// Functions/Machine Learning/F_VN_CreateLbgModel

	{attribute 'TcIecLibraryType'}
	{attribute 'external_name' := 'F_VN_CreateLbgModel_GUID_C00C428F_55C9_4971_DE2F_CFD3295E8336'}
	(* Create a LBG model of the specified type. The initial reference count is set to one if a new model is created and kept, otherwise. Models of this type neither support on-line training (sample by sample) nor retraining. *)
	FUNCTION F_VN_CreateLbgModel : HRESULT
	VAR_INPUT
		ipMlModel	:	REFERENCE TO ITcVnMlModel;	(* Returns the created model (Non-zero interface pointers are reused.) *)
		eLbgType	:	ETcVnPrototypeClusterer;	(* LBG model type *)
		nMaxClusters	:	UDINT;	(* Maximum number of clusters *)
		fMaxClusterRadius	:	LREAL;	(* Maximum allowed radius (L2 norm) of a single cluster, i.e. clusters with a higher radius will be split into smaller ones, until a global number of nMaxClusters is reached. *)
		bSingleSplitSteps	:	BOOL;	(* If true, the global optimization is always run after a single cluster has been split. If false, several clusters are split within the same step before applying the global optimization. Applying the global optimization less often is faster, but can lead to less optimal results, especially having 2 nearby clusters that could be represented by 1. *)
		hrPrev	:	HRESULT;	(* HRESULT indicating the result of previous operations (If SUCCEEDED(hrPrev) equals false, no operation is executed.) *)
	END_VAR

END_FUNCTION

// Functions/Machine Learning/F_VN_CreateLbgModelExp

	{attribute 'TcIecLibraryType'}
	{attribute 'external_name' := 'F_VN_CreateLbgModelExp_GUID_151363FF_384A_48B1_E262_C0F66CE59E70'}
	(* Create a LBG model of the specified type. The initial reference count is set to one if a new model is created and kept, otherwise. Models of this type neither support on-line training (sample by sample) nor retraining. (expert function) *)
	FUNCTION F_VN_CreateLbgModelExp : HRESULT
	VAR_INPUT
		ipMlModel	:	REFERENCE TO ITcVnMlModel;	(* Returns the created model (Non-zero interface pointers are reused.) *)
		eLbgType	:	ETcVnPrototypeClusterer;	(* LBG model type *)
		nMaxClusters	:	UDINT;	(* Maximum number of clusters *)
		fMaxClusterRadius	:	LREAL;	(* Maximum allowed radius (L2 norm) of a single cluster, i.e. clusters with a higher radius will be split into smaller ones, until a global number of nMaxClusters is reached. *)
		bSingleSplitSteps	:	BOOL;	(* If true, the global optimization is always run after a single cluster has been split. If false, several clusters are split within the same step before applying the global optimization. Applying the global optimization less often is faster, but can lead to less optimal results, especially having 2 nearby clusters that could be represented by 1. *)
		bDoublePrecision	:	BOOL;	(* If true, the model is generated with double precision (LREAL) instead of single precision (REAL). (default: FALSE) *)
		nMaxIterations	:	UDINT;	(* Maximum number of iterations (triggers the usage of the default value of 10 if it equals 0) *)
		fEpsilon	:	LREAL;	(* Maximum allowed difference of the error between two successive iterations (triggers the usage of the default value of 0.001 if it equals 0) *)
		hrPrev	:	HRESULT;	(* HRESULT indicating the result of previous operations (If SUCCEEDED(hrPrev) equals false, no operation is executed.) *)
	END_VAR

END_FUNCTION

// Functions/Machine Learning/F_VN_CreateLdaTransform

	{attribute 'TcIecLibraryType'}
	{attribute 'external_name' := 'F_VN_CreateLdaTransform_GUID_D77D3FD7_41F4_408F_DD19_2A56BE0EA5DA'}
	(* Create an LDA-based feature transform from the provided data. The number of samples must be >= the number of features and the number of classes must be >= 2. The initial reference count is set to one if a new model is created and kept, otherwise. *)
	FUNCTION F_VN_CreateLdaTransform : HRESULT
	VAR_INPUT
		ipMlModel	:	REFERENCE TO ITcVnMlModel;	(* Returns the created feature transform (Non-zero interface pointers are reused.) *)
		ipSamples	:	ITcUnknown;	(* Container holding a batch of input samples (ContainerType_Vector_Vector_REAL or ContainerType_Vector_Vector_LREAL) *)
		ipClasses	:	ITcVnContainer;	(* Class labels corresponding to the input samples (ContainerType_Vector_DINT) *)
		hrPrev	:	HRESULT;	(* HRESULT indicating the result of previous operations (If SUCCEEDED(hrPrev) equals false, no operation is executed.) *)
	END_VAR

END_FUNCTION

// Functions/Machine Learning/F_VN_CreateLdaTransformViaComponentNum

	{attribute 'TcIecLibraryType'}
	{attribute 'external_name' := 'F_VN_CreateLdaTransformViaComponentNum_GUID_F3791234_4F92_4DC1_C9F2_B56383471767'}
	(* Create an LDA-based feature transform from the provided data where the number of components to be used is predefined. The number of samples must be >= the number of features and the number of classes must be >= 2. The initial reference count is set to one if a new model is created and kept, otherwise. (expert function) *)
	FUNCTION F_VN_CreateLdaTransformViaComponentNum : HRESULT
	VAR_INPUT
		ipMlModel	:	REFERENCE TO ITcVnMlModel;	(* Returns the created feature transform (Non-zero interface pointers are reused.) *)
		ipSamples	:	ITcUnknown;	(* Container holding a batch of input samples (ContainerType_Vector_Vector_REAL or ContainerType_Vector_Vector_LREAL) *)
		ipClasses	:	ITcVnContainer;	(* Class labels corresponding to the input samples (ContainerType_Vector_DINT) *)
		nComponentNum	:	UDINT;	(* Number of components (nComponentNum must be smaller than the number of classes. A value of 0 results in the automatic computation of the maximum number of components.) *)
		hrPrev	:	HRESULT;	(* HRESULT indicating the result of previous operations (If SUCCEEDED(hrPrev) equals false, no operation is executed.) *)
	END_VAR

END_FUNCTION

// Functions/Machine Learning/F_VN_CreateNbcModel

	{attribute 'TcIecLibraryType'}
	{attribute 'external_name' := 'F_VN_CreateNbcModel_GUID_B291926B_539A_480B_CC9D_93BEFD4CDD23'}
	(* Create a normal Bayes classifier of the specified type. The initial reference count is set to one if a new model is created and kept, otherwise. In order to train normal Bayes classifiers, a sufficiently high number of samples is required for each class. It depends on the number of features and the distribution of the data. Hence, it needs to be tested for each application. Models of this type do not support on-line training (sample by sample). For the retraining of such classifier models, the set of presented classes must be identical to the previous learning steps. Otherwise, an exception is raised. *)
	FUNCTION F_VN_CreateNbcModel : HRESULT
	VAR_INPUT
		ipMlModel	:	REFERENCE TO ITcVnMlModel;	(* Returns the created model (Non-zero interface pointers are reused.) *)
		eNbcType	:	ETcVnNbc;	(* Normal Bayes classifier type *)
		hrPrev	:	HRESULT;	(* HRESULT indicating the result of previous operations (If SUCCEEDED(hrPrev) equals false, no operation is executed.) *)
	END_VAR

END_FUNCTION

// Functions/Machine Learning/F_VN_CreatePcaTransform

	{attribute 'TcIecLibraryType'}
	{attribute 'external_name' := 'F_VN_CreatePcaTransform_GUID_B2B7912B_986F_4726_FAF9_1BE1D18B6FE5'}
	(* Create a PCA-based feature transform from the provided data. The maximum number of principal components that can be computed equals the minimum of the number of samples and the number of features. The initial reference count is set to one if a new model is created and kept, otherwise. *)
	FUNCTION F_VN_CreatePcaTransform : HRESULT
	VAR_INPUT
		ipMlModel	:	REFERENCE TO ITcVnMlModel;	(* Returns the created feature transform (Non-zero interface pointers are reused.) *)
		ipSamples	:	ITcUnknown;	(* Container holding a batch of input samples (ContainerType_Vector_Vector_REAL or ContainerType_Vector_Vector_LREAL) *)
		hrPrev	:	HRESULT;	(* HRESULT indicating the result of previous operations (If SUCCEEDED(hrPrev) equals false, no operation is executed.) *)
	END_VAR

END_FUNCTION

// Functions/Machine Learning/F_VN_CreatePcaTransformViaComponentNum

	{attribute 'TcIecLibraryType'}
	{attribute 'external_name' := 'F_VN_CreatePcaTransformViaComponentNum_GUID_40831A82_3642_480F_ED98_62DA272661FF'}
	(* Create a PCA-based feature transform from the provided data where the number of prinicpal components to be used is predefined. The maximum number of principal components that can be computed equals the minimum of the number of samples and the number of features. The initial reference count is set to one if a new model is created and kept, otherwise. (expert function) *)
	FUNCTION F_VN_CreatePcaTransformViaComponentNum : HRESULT
	VAR_INPUT
		ipMlModel	:	REFERENCE TO ITcVnMlModel;	(* Returns the created feature transform (Non-zero interface pointers are reused.) *)
		ipSamples	:	ITcUnknown;	(* Container holding a batch of input samples (ContainerType_Vector_Vector_REAL or ContainerType_Vector_Vector_LREAL) *)
		nComponentNum	:	UDINT;	(* Number of principal components (A value of 0 results in the automatic computation of the maximum number of components.) *)
		hrPrev	:	HRESULT;	(* HRESULT indicating the result of previous operations (If SUCCEEDED(hrPrev) equals false, no operation is executed.) *)
	END_VAR

END_FUNCTION

// Functions/Machine Learning/F_VN_CreatePcaTransformViaVariance

	{attribute 'TcIecLibraryType'}
	{attribute 'external_name' := 'F_VN_CreatePcaTransformViaVariance_GUID_7593ED13_6826_4CA8_C043_9ACE9956F61F'}
	(* Create a PCA-based feature transform from the provided data based on a given fraction of variance to be retained. The maximum number of principal components that can be computed equals the minimum of the number of samples and the number of features. The initial reference count is set to one if a new model is created and kept, otherwise. (expert function) *)
	FUNCTION F_VN_CreatePcaTransformViaVariance : HRESULT
	VAR_INPUT
		ipMlModel	:	REFERENCE TO ITcVnMlModel;	(* Returns the created feature transform (Non-zero interface pointers are reused.) *)
		ipSamples	:	ITcUnknown;	(* Container holding a batch of input samples (ContainerType_Vector_Vector_REAL or ContainerType_Vector_Vector_LREAL) *)
		fRetainedVariance	:	LREAL;	(* Fraction of variance that is to be retained by the PCA (A value of 1.0 signifies 100%.) *)
		hrPrev	:	HRESULT;	(* HRESULT indicating the result of previous operations (If SUCCEEDED(hrPrev) equals false, no operation is executed.) *)
	END_VAR

END_FUNCTION

// Functions/Machine Learning/F_VN_CreateRTreesModel

	{attribute 'TcIecLibraryType'}
	{attribute 'external_name' := 'F_VN_CreateRTreesModel_GUID_361E493C_0B92_4424_E04B_1ECB2685F6EE'}
	(* Create a random trees model of the specified type. The initial reference count is set to one if a new model is created and kept, otherwise. Models of this type neither support on-line training (sample by sample) nor retraining. Predictions can only be scalar. *)
	FUNCTION F_VN_CreateRTreesModel : HRESULT
	VAR_INPUT
		ipMlModel	:	REFERENCE TO ITcVnMlModel;	(* Returns the created model (Non-zero interface pointers are reused.) *)
		eRTreesType	:	ETcVnRTrees;	(* Random trees model type *)
		hrPrev	:	HRESULT;	(* HRESULT indicating the result of previous operations (If SUCCEEDED(hrPrev) equals false, no operation is executed.) *)
	END_VAR

END_FUNCTION

// Functions/Machine Learning/F_VN_CreateRTreesModelExp

	{attribute 'TcIecLibraryType'}
	{attribute 'external_name' := 'F_VN_CreateRTreesModelExp_GUID_DCAA6B97_3E63_4846_D44A_21B2790A7B88'}
	(* Create a random trees model of the specified type. The initial reference count is set to one if a new model is created and kept, otherwise. Models of this type neither support on-line training (sample by sample) nor retraining. Predictions can only be scalar. (expert function) *)
	FUNCTION F_VN_CreateRTreesModelExp : HRESULT
	VAR_INPUT
		ipMlModel	:	REFERENCE TO ITcVnMlModel;	(* Returns the created model (Non-zero interface pointers are reused.) *)
		eRTreesType	:	ETcVnRTrees;	(* Random trees model type *)
		nMaxDepth	:	UDINT;	(* Maximum tree depth (default: 5) *)
		nMinSamples	:	UDINT;	(* Minimum number of samples within a node required for splitting (default: 10) *)
		nActiveVariables	:	UDINT;	(* Number of variables considered for splitting (0 means sqrt(total number of variables); default: 0) *)
		nMaxIterations	:	UDINT;	(* Maximum number of iterations (disabled if it equals 0 and fEpsilon is different from 0.0; triggers the usage of the default value of 50 if nMaxIterations and fEpsilon equal 0) *)
		fEpsilon	:	LREAL;	(* Maximum allowed difference of the error between two successive iterations (disabled if it equals 0.0 and nMaxIterations is different from 0; triggers the usage of the default value of 0.1 if nMaxIterations and fEpsilon equal 0) *)
		hrPrev	:	HRESULT;	(* HRESULT indicating the result of previous operations (If SUCCEEDED(hrPrev) equals false, no operation is executed.) *)
	END_VAR

END_FUNCTION

// Functions/Machine Learning/F_VN_CreateRTreesModelExp2

	{attribute 'TcIecLibraryType'}
	{attribute 'external_name' := 'F_VN_CreateRTreesModelExp2_GUID_A3B951DB_7DFC_4984_C9A1_23F5FD764134'}
	(* Create a random trees model of the specified type. The initial reference count is set to one if a new model is created and kept, otherwise. Models of this type neither support on-line training (sample by sample) nor retraining. Predictions can only be scalar. (expert function) *)
	FUNCTION F_VN_CreateRTreesModelExp2 : HRESULT
	VAR_INPUT
		ipMlModel	:	REFERENCE TO ITcVnMlModel;	(* Returns the created model (Non-zero interface pointers are reused.) *)
		eRTreesType	:	ETcVnRTrees;	(* Random trees model type *)
		nMaxDepth	:	UDINT;	(* Maximum tree depth (default: 5) *)
		nMinSamples	:	UDINT;	(* Minimum number of samples within a node required for splitting (default: 10) *)
		nActiveVariables	:	UDINT;	(* Number of variables considered for splitting (0 means sqrt(total number of variables); default: 0) *)
		nMaxIterations	:	UDINT;	(* Maximum number of iterations (disabled if it equals 0 and fEpsilon is different from 0.0; triggers the usage of the default value of 50 if nMaxIterations and fEpsilon equal 0) *)
		fEpsilon	:	LREAL;	(* Maximum allowed difference of the error between two successive iterations (disabled if it equals 0.0 and nMaxIterations is different from 0; triggers the usage of the default value of 0.1 if nMaxIterations and fEpsilon equal 0) *)
		fRegressionAccuracy	:	REAL;	(* Termination criterion for regressors (only for regressors; set to default if not allowed; default: 0.0) *)
		ipClassPriors	:	ITcVnContainer;	(* Class priors (ContainerType_Vector_REAL or ContainerType_Vector_LREAL; only for classifiers; optional, set to 0 if not required or not allowed; default: 0) *)
		hrPrev	:	HRESULT;	(* HRESULT indicating the result of previous operations (If SUCCEEDED(hrPrev) equals false, no operation is executed.) *)
	END_VAR

END_FUNCTION

// Functions/Machine Learning/F_VN_CreateStaModel

	{attribute 'TcIecLibraryType'}
	{attribute 'external_name' := 'F_VN_CreateStaModel_GUID_0E65F544_36C9_4DC3_E430_89B77157AED0'}
	(* Create a Simplified TopoART neural network of the specified type. The initial reference count is set to one if a new model is created and kept, otherwise. Models of this type support on-line training (sample by sample), retraining, as well as scalar and vectorial predictions. It requires all input except class labels (i.e., samples and training outputs/predictions) to lie in the interval [0.0, 1.0]. The predictions of regressors need to be rescaled from the interval [0.0, 1.0] to their respective value range before usage. Depending on the parameter settings and the number of available training samples, repeated training with the same data may improve the results. Like other neural networks based on the Adaptive Resonance Theory (ART), Simplified TopoART neural networks are not prone to catastrophic inference and patricularly well-suited to incremental learning tasks. *)
	FUNCTION F_VN_CreateStaModel : HRESULT
	VAR_INPUT
		ipMlModel	:	REFERENCE TO ITcVnMlModel;	(* Returns the created model (Non-zero interface pointers are reused.) *)
		eStaType	:	ETcVnSta;	(* Simpified TopoART model type *)
		fRho	:	LREAL;	(* Vigilance parameter (controls the number of neurons that are inserted and the maximum size of the formed categories; valid range: [0.0, 1.0]; suggested range: [0.8, 1.0)) *)
		hrPrev	:	HRESULT;	(* HRESULT indicating the result of previous operations (If SUCCEEDED(hrPrev) equals false, no operation is executed.) *)
	END_VAR

END_FUNCTION

// Functions/Machine Learning/F_VN_CreateStaModelExp

	{attribute 'TcIecLibraryType'}
	{attribute 'external_name' := 'F_VN_CreateStaModelExp_GUID_60C95C96_C531_4303_F18A_D4FE39CB265F'}
	(* Create a Simplified TopoART neural network of the specified type. The initial reference count is set to one if a new model is created and kept, otherwise. Models of this type support on-line training (sample by sample), retraining, as well as scalar and vectorial predictions. It requires all input except class labels (i.e., samples and training outputs/predictions) to lie in the interval [0.0, 1.0]. The predictions of regressors need to be rescaled from the interval [0.0, 1.0] to their respective value range before usage. Depending on the parameter settings and the number of available training samples, repeated training with the same data may improve the results. Like other neural networks based on the Adaptive Resonance Theory (ART), Simplified TopoART neural networks are not prone to catastrophic inference and patricularly well-suited to incremental learning tasks. (expert function) *)
	FUNCTION F_VN_CreateStaModelExp : HRESULT
	VAR_INPUT
		ipMlModel	:	REFERENCE TO ITcVnMlModel;	(* Returns the created model (Non-zero interface pointers are reused.) *)
		eStaType	:	ETcVnSta;	(* Simpified TopoART model type *)
		fRho	:	LREAL;	(* Vigilance parameter (controls the number of neurons that are inserted and the maximum size of the formed categories; valid range: [0.0, 1.0]; suggested range: [0.8, 1.0)) *)
		nNu	:	UDINT;	(* Number of neurons used for classification and prediction (must be larger than or equal to 1; suggested range: [1, 10); default: 3) *)
		bDoublePrecision	:	BOOL;	(* If true, the model is generated with double precision (LREAL) instead of single precision (REAL). (default: FALSE) *)
		hrPrev	:	HRESULT;	(* HRESULT indicating the result of previous operations (If SUCCEEDED(hrPrev) equals false, no operation is executed.) *)
	END_VAR

END_FUNCTION

// Functions/Machine Learning/F_VN_CreateStaModelExp2

	{attribute 'TcIecLibraryType'}
	{attribute 'external_name' := 'F_VN_CreateStaModelExp2_GUID_DC5ABDD2_E185_452E_E9B5_8EF979CD80B8'}
	(* Create a Simplified TopoART neural network of the specified type. The initial reference count is set to one if a new model is created and kept, otherwise. Models of this type support on-line training (sample by sample), retraining, as well as scalar and vectorial predictions. It requires all input except class labels (i.e., samples and training outputs/predictions) to lie in the interval [0.0, 1.0]. The predictions of regressors need to be rescaled from the interval [0.0, 1.0] to their respective value range before usage. Depending on the parameter settings and the number of available training samples, repeated training with the same data may improve the results. Like other neural networks based on the Adaptive Resonance Theory (ART), Simplified TopoART neural networks are not prone to catastrophic inference and patricularly well-suited to incremental learning tasks. (additional expert function providing parameters for fine-tuning and noise reduction) *)
	FUNCTION F_VN_CreateStaModelExp2 : HRESULT
	VAR_INPUT
		ipMlModel	:	REFERENCE TO ITcVnMlModel;	(* Returns the created model (Non-zero interface pointers are reused.) *)
		eStaType	:	ETcVnSta;	(* Simpified TopoART model type *)
		fRho	:	LREAL;	(* Vigilance parameter (controls the number of neurons that are inserted and the maximum size of the formed categories; valid range: [0.0, 1.0]; suggested range: [0.8, 1.0)) *)
		nNu	:	UDINT;	(* Number of neurons used for classification and prediction (must be larger than or equal to 1; suggested range: [1, 10); default: 3) *)
		bDoublePrecision	:	BOOL;	(* If true, the model is generated with double precision (LREAL) instead of single precision (REAL). (default: FALSE) *)
		fBetaSbm	:	LREAL;	(* Learning rate of the second best-matching neuron (learning the second best-matching neuron keeps related categories closer together and might improve the results but may require a higher number of neurons and training runs; a value of 0.0 disables learning of the second best-matching neuron; valid range: [0.0, 1.0]; suggested range: [0.0, 0.5]); default: 0.0 *)
		nPhi	:	UDINT;	(* Number of samples a neuron must have learnt to become permanent (required for noise reduction; works in conjunction with nTau; must be larger than or equal to 1; higher values intensify noise reduction; a value of 1 disables removal of neuron candidates; default: 1) *)
		nTau	:	UDINT;	(* Number of learning steps after which node removal is performed (required for noise reduction; works in conjunction with nPhi; must be large enough to allow neuron candidates representing non-noise samples to become the best-matching neuron at least nPhi times before node removal; default: 100) *)
		hrPrev	:	HRESULT;	(* HRESULT indicating the result of previous operations (If SUCCEEDED(hrPrev) equals false, no operation is executed.) *)
	END_VAR

END_FUNCTION

// Functions/Machine Learning/F_VN_CreateSvmModel

	{attribute 'TcIecLibraryType'}
	{attribute 'external_name' := 'F_VN_CreateSvmModel_GUID_6608170F_8E55_4CB7_CA5D_A5F69CCA9D00'}
	(* Create an SVM model of the specified type. The initial reference count is set to one if a new model is created and kept, otherwise. Models of this type neither support on-line training (sample by sample) nor retraining. Predictions can only be scalar. *)
	FUNCTION F_VN_CreateSvmModel : HRESULT
	VAR_INPUT
		ipMlModel	:	REFERENCE TO ITcVnMlModel;	(* Returns the created model (Non-zero interface pointers are reused.) *)
		eSvmType	:	ETcVnSvm;	(* SVM model type *)
		fC	:	LREAL;	(* Parameter C (required for TCVN_SVM_C_CLASSIFIER, TCVN_SVM_EPS_REGRESSOR, and TCVN_SVM_NU_REGRESSOR; ignored otherwise) *)
		fNu	:	LREAL;	(* Parameter nu (required for TCVN_SVM_NU_CLASSIFIER, TCVN_SVM_NOVELTY_DETECTOR, and TCVN_SVM_NU_REGRESSOR; ignored otherwise) *)
		fP	:	LREAL;	(* Parameter p (required for TCVN_SVM_EPS_REGRESSOR; ignored otherwise) *)
		eKernelType	:	ETcVnSvmKernelType;	(* Kernel type *)
		fGamma	:	LREAL;	(* Parameter gamma (used by polynomial, RBF, sigmoid, and chi-squared kernels; ignored otherwise) *)
		fCoef0	:	LREAL;	(* parameter coef0 (used by polynomial and sigmoid kernels; ignored otherwise) *)
		fDegree	:	LREAL;	(* Degree (used by polynomial kernels; ignored otherwise) *)
		hrPrev	:	HRESULT;	(* HRESULT indicating the result of previous operations (If SUCCEEDED(hrPrev) equals false, no operation is executed.) *)
	END_VAR

END_FUNCTION

// Functions/Machine Learning/F_VN_CreateSvmModelExp

	{attribute 'TcIecLibraryType'}
	{attribute 'external_name' := 'F_VN_CreateSvmModelExp_GUID_6B1D8D00_DDAB_4438_FB92_B0FDD976C945'}
	(* Create an SVM model of the specified type. The initial reference count is set to one if a new model is created and kept, otherwise. Models of this type neither support on-line training (sample by sample) nor retraining. Predictions can only be scalar. (expert function) *)
	FUNCTION F_VN_CreateSvmModelExp : HRESULT
	VAR_INPUT
		ipMlModel	:	REFERENCE TO ITcVnMlModel;	(* Returns the created model (Non-zero interface pointers are reused.) *)
		eSvmType	:	ETcVnSvm;	(* SVM model type *)
		fC	:	LREAL;	(* Parameter C (required for TCVN_SVM_C_CLASSIFIER, TCVN_SVM_EPS_REGRESSOR, and TCVN_SVM_NU_REGRESSOR; ignored otherwise) *)
		fNu	:	LREAL;	(* Parameter nu (required for TCVN_SVM_NU_CLASSIFIER, TCVN_SVM_NOVELTY_DETECTOR, and TCVN_SVM_NU_REGRESSOR; ignored otherwise) *)
		fP	:	LREAL;	(* Parameter p (required for TCVN_SVM_EPS_REGRESSOR; ignored otherwise) *)
		eKernelType	:	ETcVnSvmKernelType;	(* Kernel type *)
		fGamma	:	LREAL;	(* Parameter gamma (used by polynomial, RBF, sigmoid, and chi-squared kernels; ignored otherwise) *)
		fCoef0	:	LREAL;	(* Parameter coef0 (used by polynomial and sigmoid kernels; ignored otherwise) *)
		fDegree	:	LREAL;	(* Degree (used by polynomial kernels; ignored otherwise) *)
		nMaxIterations	:	UDINT;	(* Maximum number of iterations (disabled if it equals 0 and fEpsilon is different from 0.0; triggers the usage of the default value of 100000 if nMaxIterations and fEpsilon equal 0) *)
		fEpsilon	:	LREAL;	(* Maximum allowed difference of the error between two successive iterations (disabled if it equals 0.0 and nMaxIterations is different from 0; triggers the usage of the default value of 0.00001 if nMaxIterations and fEpsilon equal 0) *)
		hrPrev	:	HRESULT;	(* HRESULT indicating the result of previous operations (If SUCCEEDED(hrPrev) equals false, no operation is executed.) *)
	END_VAR

END_FUNCTION

// Functions/Machine Learning/F_VN_CreateSvmModelExp2

	{attribute 'TcIecLibraryType'}
	{attribute 'external_name' := 'F_VN_CreateSvmModelExp2_GUID_6FD5F0B0_2D5E_4EC3_E8E4_B31A19CD0010'}
	(* Create an SVM model of the specified type. The initial reference count is set to one if a new model is created and kept, otherwise. Models of this type neither support on-line training (sample by sample) nor retraining. Predictions can only be scalar. (additional expert function for C support vector classifiers) *)
	FUNCTION F_VN_CreateSvmModelExp2 : HRESULT
	VAR_INPUT
		ipMlModel	:	REFERENCE TO ITcVnMlModel;	(* Returns the created model (Non-zero interface pointers are reused.) *)
		eSvmType	:	ETcVnSvm;	(* SVM model type *)
		fC	:	LREAL;	(* Parameter C (required for TCVN_SVM_C_CLASSIFIER, TCVN_SVM_EPS_REGRESSOR, and TCVN_SVM_NU_REGRESSOR; ignored otherwise) *)
		fNu	:	LREAL;	(* Parameter nu (required for TCVN_SVM_NU_CLASSIFIER, TCVN_SVM_NOVELTY_DETECTOR, and TCVN_SVM_NU_REGRESSOR; ignored otherwise) *)
		fP	:	LREAL;	(* Parameter p (required for TCVN_SVM_EPS_REGRESSOR; ignored otherwise) *)
		eKernelType	:	ETcVnSvmKernelType;	(* Kernel type *)
		fGamma	:	LREAL;	(* Parameter gamma (used by polynomial, RBF, sigmoid, and chi-squared kernels; ignored otherwise) *)
		fCoef0	:	LREAL;	(* Parameter coef0 (used by polynomial and sigmoid kernels; ignored otherwise) *)
		fDegree	:	LREAL;	(* Degree (used by polynomial kernels; ignored otherwise) *)
		nMaxIterations	:	UDINT;	(* Maximum number of iterations (disabled if it equals 0 and fEpsilon is different from 0.0; triggers the usage of the default value of 100000 if nMaxIterations and fEpsilon equal 0) *)
		fEpsilon	:	LREAL;	(* Maximum allowed difference of the error between two successive iterations (disabled if it equals 0.0 and nMaxIterations is different from 0; triggers the usage of the default value of 0.00001 if nMaxIterations and fEpsilon equal 0) *)
		ipClassWeights	:	ITcVnContainer;	(* Class weights (ContainerType_Vector_REAL or ContainerType_Vector_LREAL; only valid if eSvmType equals TCVN_SVM_C_CLASSIFIER; optional, set to 0 if not required or not allowed; default: 0) *)
		hrPrev	:	HRESULT;	(* HRESULT indicating the result of previous operations (If SUCCEEDED(hrPrev) equals false, no operation is executed.) *)
	END_VAR

END_FUNCTION

// Functions/Machine Learning/F_VN_CreateSvmSgdClassifier

	{attribute 'TcIecLibraryType'}
	{attribute 'external_name' := 'F_VN_CreateSvmSgdClassifier_GUID_C9EE268D_C05A_48F3_D32E_D9B3E0FBCDCB'}
	(* Create a linear SVM classifier using stochastic gradient descent for training. The initial reference count is set to one if a new model is created and kept, otherwise. This SVM classifier is only applicable to binary classification problems. It learns a separating hyperplane between a class with label -1 and a class with label 1. These class labels are predefined. For training, any positive class labels are mapped to 1 and any negative class labels are mapped to -1. Models of this type neither support on-line training (sample by sample) nor retraining. *)
	FUNCTION F_VN_CreateSvmSgdClassifier : HRESULT
	VAR_INPUT
		ipMlModel	:	REFERENCE TO ITcVnMlModel;	(* Returns the created model (Non-zero interface pointers are reused.) *)
		hrPrev	:	HRESULT;	(* HRESULT indicating the result of previous operations (If SUCCEEDED(hrPrev) equals false, no operation is executed.) *)
	END_VAR

END_FUNCTION

// Functions/Machine Learning/F_VN_CreateSvmSgdClassifierExp

	{attribute 'TcIecLibraryType'}
	{attribute 'external_name' := 'F_VN_CreateSvmSgdClassifierExp_GUID_35712FDB_BBEA_4B29_FC4D_61FC511DA0EB'}
	(* Create a linear SVM classifier using stochastic gradient descent for training. The initial reference count is set to one if a new model is created and kept, otherwise. This SVM classifier is only applicable to binary classification problems. It learns a separating hyperplane between a class with label -1 and a class with label 1. These class labels are predefined. For training, any positive class labels are mapped to 1 and any negative class labels are mapped to -1. Models of this type neither support on-line training (sample by sample) nor retraining. (expert function) *)
	FUNCTION F_VN_CreateSvmSgdClassifierExp : HRESULT
	VAR_INPUT
		ipMlModel	:	REFERENCE TO ITcVnMlModel;	(* Returns the created model (Non-zero interface pointers are reused.) *)
		eType	:	ETcVnSvmSgdClassifierType;	(* Learning algorithm type (default: TCVN_SSCT_ASGD) *)
		eMarginType	:	ETcVnSvmSgdClassifierMarginType;	(* Margin type (default: TCVN_SSCMT_SOFT_MARGIN) *)
		fMarginRegularization	:	REAL;	(* Margin regularization parameter (default: 0.00001) *)
		fInitialStepSize	:	REAL;	(* Initial step size (default: 0.05) *)
		fStepDecreasingPower	:	REAL;	(* Power parameter (default: 0.75) *)
		nMaxIterations	:	UDINT;	(* Maximum number of iterations (disabled if it equals 0 and fEpsilon is different from 0.0; triggers the usage of the default value of 100000 if nMaxIterations and fEpsilon equal 0) *)
		fEpsilon	:	LREAL;	(* Maximum allowed difference of the error between two successive iterations (disabled if it equals 0.0 and nMaxIterations is different from 0; triggers the usage of the default value of 0.00001 if nMaxIterations and fEpsilon equal 0) *)
		hrPrev	:	HRESULT;	(* HRESULT indicating the result of previous operations (If SUCCEEDED(hrPrev) equals false, no operation is executed.) *)
	END_VAR

END_FUNCTION

// Functions/Machine Learning/F_VN_FeatureTransform

	{attribute 'TcIecLibraryType'}
	{attribute 'external_name' := 'F_VN_FeatureTransform_GUID_C607A85C_BB4D_46AF_DE31_007EC6E109EA'}
	(* Apply a feature transform to one or more sample(s). *)
	FUNCTION F_VN_FeatureTransform : HRESULT
	VAR_INPUT
		ipFeatureTransform	:	ITcVnMlModel;	(* Feature transform instance to be used *)
		ipSamples	:	ITcUnknown;	(* Container holding one or more of input sample(s) (ContainerType_Vector_REAL, ContainerType_Vector_LREAL, ContainerType_Vector_Vector_REAL, or ContainerType_Vector_Vector_LREAL) *)
		pipTransformed	:	POINTER TO ITcUnknown;	(* Returns the transformed sample(s) using the same type like ipSamples *)
		hrPrev	:	HRESULT;	(* HRESULT indicating the result of previous operations (If SUCCEEDED(hrPrev) equals false, no operation is executed.) *)
	END_VAR

END_FUNCTION

// Functions/Machine Learning/F_VN_GetBatchClusters

	{attribute 'TcIecLibraryType'}
	{attribute 'external_name' := 'F_VN_GetBatchClusters_GUID_528E2B3F_88E6_4E83_EA33_7AE81270B54C'}
	(* Get the IDs of the best-matching clusters of a batch of samples. *)
	FUNCTION F_VN_GetBatchClusters : HRESULT
	VAR_INPUT
		ipClusterer	:	ITcVnMlModel;	(* Clusterer to be used *)
		ipSamples	:	ITcUnknown;	(* Container holding a batch of input samples (ContainerType_Vector_Vector_REAL or ContainerType_Vector_Vector_LREAL) *)
		ipClusters	:	REFERENCE TO ITcVnContainer;	(* Returns the cluster IDs (ContainerType_Vector_DINT) *)
		hrPrev	:	HRESULT;	(* HRESULT indicating the result of previous operations (If SUCCEEDED(hrPrev) equals false, no operation is executed.) *)
	END_VAR

END_FUNCTION

// Functions/Machine Learning/F_VN_GetBatchClustersExp

	{attribute 'TcIecLibraryType'}
	{attribute 'external_name' := 'F_VN_GetBatchClustersExp_GUID_EA27BC56_5775_49D6_D10F_C11E25D16558'}
	(* Get the IDs of the best-matching clusters of a batch of samples. *)
	FUNCTION F_VN_GetBatchClustersExp : HRESULT
	VAR_INPUT
		ipClusterer	:	ITcVnMlModel;	(* Clusterer to be used *)
		ipSamples	:	ITcUnknown;	(* Container holding a batch of input samples (ContainerType_Vector_Vector_REAL or ContainerType_Vector_Vector_LREAL) *)
		ipClusters	:	REFERENCE TO ITcVnContainer;	(* Returns the cluster IDs (ContainerType_Vector_DINT) *)
		ipNovelties	:	REFERENCE TO ITcVnContainer;	(* Returns the degree of novelty (0.0 if a sample is completely known; > 0.0 otherwise) of each sample (ContainerType_Vector_REAL; optional, set to 0 if not required) *)
		hrPrev	:	HRESULT;	(* HRESULT indicating the result of previous operations (If SUCCEEDED(hrPrev) equals false, no operation is executed.) *)
	END_VAR

END_FUNCTION

// Functions/Machine Learning/F_VN_GetBatchNovelties

	{attribute 'TcIecLibraryType'}
	{attribute 'external_name' := 'F_VN_GetBatchNovelties_GUID_7C3BAC31_B33D_4380_E65E_AEEC8DBAEDE0'}
	(* Get the degree of novelty of multiple samples. *)
	FUNCTION F_VN_GetBatchNovelties : HRESULT
	VAR_INPUT
		ipNoveltyDetector	:	ITcVnMlModel;	(* Novelty detector to be used *)
		ipSamples	:	ITcUnknown;	(* Container holding a batch of input samples (ContainerType_Vector_Vector_REAL or ContainerType_Vector_Vector_LREAL) *)
		ipNovelties	:	REFERENCE TO ITcVnContainer;	(* Returns the degree of novelty (0.0 if a sample is completely known; > 0.0 otherwise) of each sample (ContainerType_Vector_REAL) *)
		hrPrev	:	HRESULT;	(* HRESULT indicating the result of previous operations (If SUCCEEDED(hrPrev) equals false, no operation is executed.) *)
	END_VAR

END_FUNCTION

// Functions/Machine Learning/F_VN_GetClusterCenter

	{attribute 'TcIecLibraryType'}
	{attribute 'external_name' := 'F_VN_GetClusterCenter_GUID_0F8CBC11_259F_42B1_EE6F_9AD92F7A06AE'}
	(* Get the center of a cluster. *)
	FUNCTION F_VN_GetClusterCenter : HRESULT
	VAR_INPUT
		ipClusterer	:	ITcVnMlModel;	(* Clusterer to be used *)
		nCluster	:	DINT;	(* Cluster ID of the cluster the center of which is requested *)
		ipCenter	:	REFERENCE TO ITcVnContainer;	(* Returns the cluster center (ContainerType_Vector_REAL or ContainerType_Vector_LREAL depending on the floating point type internally used by the clusterer) *)
		hrPrev	:	HRESULT;	(* HRESULT indicating the result of previous operations (If SUCCEEDED(hrPrev) equals false, no operation is executed.) *)
	END_VAR

END_FUNCTION

// Functions/Machine Learning/F_VN_GetClusterNum

	{attribute 'TcIecLibraryType'}
	{attribute 'external_name' := 'F_VN_GetClusterNum_GUID_548F7E1B_5B12_494E_CC7F_3482B1B8572D'}
	(* Get the number of clusters used by this clusterer. *)
	FUNCTION F_VN_GetClusterNum : HRESULT
	VAR_INPUT
		ipClusterer	:	ITcVnMlModel;	(* Clusterer to be used *)
	END_VAR
	VAR_IN_OUT
		nClusterNum	:	ULINT;	(* Returns the number of clusters *)
	END_VAR
	VAR_INPUT
		hrPrev	:	HRESULT;	(* HRESULT indicating the result of previous operations (If SUCCEEDED(hrPrev) equals false, no operation is executed.) *)
	END_VAR

END_FUNCTION

// Functions/Machine Learning/F_VN_GetFeatureScales

	{attribute 'TcIecLibraryType'}
	{attribute 'external_name' := 'F_VN_GetFeatureScales_GUID_FE369AE1_304E_4286_ECEF_EB86184B6B22'}
	(* Calculate the scaling parameters for each feature in the input samples based on the scaling type. *)
	FUNCTION F_VN_GetFeatureScales : HRESULT
	VAR_INPUT
		ipSamples	:	ITcVnContainer;	(* Container holding input sample(s) (ContainerType_Vector_REAL, ContainerType_Vector_LREAL, ContainerType_Vector_Vector_REAL or ContainerType_Vector_Vector_LREAL) *)
		ipScales	:	REFERENCE TO ITcVnContainer;	(* Returns a container with the scaling parameters for each feature (Vector_REAL or Vector_LREAL depending on the type of ipSamples). *)
		eFeatureScalingType	:	ETcVnFeatureScalingType;	(* Feature scaling type *)
		hrPrev	:	HRESULT;	(* HRESULT indicating the result of previous operations (If SUCCEEDED(hrPrev) equals false, no operation is executed.) *)
	END_VAR

END_FUNCTION

// Functions/Machine Learning/F_VN_GetSampleCluster

	{attribute 'TcIecLibraryType'}
	{attribute 'external_name' := 'F_VN_GetSampleCluster_GUID_32F204F3_A186_4B1B_F32F_2AD94C5430BB'}
	(* Get the ID of the best-matching cluster of a single sample. *)
	FUNCTION F_VN_GetSampleCluster : HRESULT
	VAR_INPUT
		ipClusterer	:	ITcVnMlModel;	(* Clusterer to be used *)
		ipSample	:	ITcUnknown;	(* Container holding a single input sample (ContainerType_Vector_REAL or ContainerType_Vector_LREAL) *)
	END_VAR
	VAR_IN_OUT
		nCluster	:	DINT;	(* Returns the ID of the cluster the sample has been assigned to *)
	END_VAR
	VAR_INPUT
		hrPrev	:	HRESULT;	(* HRESULT indicating the result of previous operations (If SUCCEEDED(hrPrev) equals false, no operation is executed.) *)
	END_VAR

END_FUNCTION

// Functions/Machine Learning/F_VN_GetSampleClusterExp

	{attribute 'TcIecLibraryType'}
	{attribute 'external_name' := 'F_VN_GetSampleClusterExp_GUID_3477724D_EC43_4000_ECAE_3FA8E7C5B7E6'}
	(* Get the ID of the best-matching cluster of a single sample. (expert function) *)
	FUNCTION F_VN_GetSampleClusterExp : HRESULT
	VAR_INPUT
		ipClusterer	:	ITcVnMlModel;	(* Clusterer to be used *)
		ipSample	:	ITcUnknown;	(* Container holding a single input sample (ContainerType_Vector_REAL or ContainerType_Vector_LREAL) *)
	END_VAR
	VAR_IN_OUT
		nCluster	:	DINT;	(* Returns the ID of the cluster the sample has been assigned to *)
	END_VAR
	VAR_INPUT
		fNovelty	:	REFERENCE TO REAL;	(* Returns the degree of novelty (0.0 if a sample is completely known; > 0.0 otherwise) of the presented sample (optional, set to 0 if not required) *)
		hrPrev	:	HRESULT;	(* HRESULT indicating the result of previous operations (If SUCCEEDED(hrPrev) equals false, no operation is executed.) *)
	END_VAR

END_FUNCTION

// Functions/Machine Learning/F_VN_GetSampleNovelty

	{attribute 'TcIecLibraryType'}
	{attribute 'external_name' := 'F_VN_GetSampleNovelty_GUID_D2B7DAC3_715A_4874_EE3F_A314571BD5C4'}
	(* Get the degree of novelty of a single sample. *)
	FUNCTION F_VN_GetSampleNovelty : HRESULT
	VAR_INPUT
		ipNoveltyDetector	:	ITcVnMlModel;	(* Novelty detector to be used *)
		ipSample	:	ITcUnknown;	(* Container holding a single input sample (ContainerType_Vector_REAL or ContainerType_Vector_LREAL) *)
	END_VAR
	VAR_IN_OUT
		fNovelty	:	REAL;	(* Returns the degree of novelty (0.0 if a sample is completely known; > 0.0 otherwise) of the presented sample *)
	END_VAR
	VAR_INPUT
		hrPrev	:	HRESULT;	(* HRESULT indicating the result of previous operations (If SUCCEEDED(hrPrev) equals false, no operation is executed.) *)
	END_VAR

END_FUNCTION

// Functions/Machine Learning/F_VN_InverseFeatureScaling

	{attribute 'TcIecLibraryType'}
	{attribute 'external_name' := 'F_VN_InverseFeatureScaling_GUID_15907737_CCFF_4C4C_EA62_BDD72702354F'}
	(* Apply the inverse of feature scaling to one or more sample(s). *)
	FUNCTION F_VN_InverseFeatureScaling : HRESULT
	VAR_INPUT
		ipSamples	:	ITcVnContainer;	(* Container holding one or more input sample(s) (ContainerType_Vector_REAL, ContainerType_Vector_LREAL, ContainerType_Vector_Vector_REAL, or ContainerType_Vector_Vector_LREAL) *)
		ipScales	:	ITcVnContainer;	(* Container with the scaling parameters of each feature (type ContainerType_Vector_REAL or ContainerType_Vector_LREAL). *)
		ipInverseSamples	:	REFERENCE TO ITcVnContainer;	(* Returns the inversed sample(s) using the scaling type and parameters of ipScales. It has the same type of ipSamples. If the same container ipSamples is used, the source data will be replaced. *)
		hrPrev	:	HRESULT;	(* HRESULT indicating the result of previous operations (If SUCCEEDED(hrPrev) equals false, no operation is executed.) *)
	END_VAR

END_FUNCTION

// Functions/Machine Learning/F_VN_InverseFeatureScaling_REAL

	{attribute 'TcIecLibraryType'}
	{attribute 'external_name' := 'F_VN_InverseFeatureScaling_REAL_GUID_F91E68ED_D57C_4247_F2CE_BAB31E6A8058'}
	(* Apply the inverse of feature scaling to a single value. *)
	FUNCTION F_VN_InverseFeatureScaling_REAL : HRESULT
	VAR_INPUT
		fSample	:	REAL;	(* Sample value *)
		ipScales	:	ITcVnContainer;	(* Container with the scaling parameters of each feature (type ContainerType_Vector_REAL or ContainerType_Vector_LREAL). *)
	END_VAR
	VAR_IN_OUT
		fInverseSample	:	REAL;	(* Returns the inversed sample. *)
	END_VAR
	VAR_INPUT
		hrPrev	:	HRESULT;	(* HRESULT indicating the result of previous operations (If SUCCEEDED(hrPrev) equals false, no operation is executed.) *)
	END_VAR

END_FUNCTION

// Functions/Machine Learning/F_VN_InverseFeatureScalingExp

	{attribute 'TcIecLibraryType'}
	{attribute 'external_name' := 'F_VN_InverseFeatureScalingExp_GUID_8B0E0F8E_1465_40CF_D892_BBD7360C8D03'}
	(* Apply the inverse of feature scaling to one or more sample(s). [fA, fB] should be used if the scaling has been performed using TCVN_FST1_MINMAX with a predetermined output range.. (expert function) *)
	FUNCTION F_VN_InverseFeatureScalingExp : HRESULT
	VAR_INPUT
		ipSamples	:	ITcVnContainer;	(* Container holding one or more input sample(s) (ContainerType_Vector_REAL, ContainerType_Vector_LREAL, ContainerType_Vector_Vector_REAL, or ContainerType_Vector_Vector_LREAL) *)
		ipScales	:	ITcVnContainer;	(* Container with the scaling parameters of each feature (type ContainerType_Vector_REAL or ContainerType_Vector_LREAL). *)
		ipInverseSamples	:	REFERENCE TO ITcVnContainer;	(* Returns the inversed sample(s) using the scaling type and parameters of ipScales. It has the same type of ipSamples. If the same container ipSamples is used, the source data will be replaced. *)
		fA	:	LREAL;	(* represents the lower bound of the range for TCVN_FST1_MINMAX *)
		fB	:	LREAL;	(* represents the upper bound of the range for TCVN_FST1_MINMAX *)
		hrPrev	:	HRESULT;	(* HRESULT indicating the result of previous operations (If SUCCEEDED(hrPrev) equals false, no operation is executed.) *)
	END_VAR

END_FUNCTION

// Functions/Machine Learning/F_VN_InverseFeatureScalingExp_REAL

	{attribute 'TcIecLibraryType'}
	{attribute 'external_name' := 'F_VN_InverseFeatureScalingExp_REAL_GUID_22A89423_ED3D_4292_D684_932CEE57D3B8'}
	(* Apply the inverse of feature scaling to a single value. [fA, fB] should be used if the scaling has been performed using TCVN_FST1_MINMAX with a predetermined output range. *)
	FUNCTION F_VN_InverseFeatureScalingExp_REAL : HRESULT
	VAR_INPUT
		fSample	:	REAL;	(* Sample value *)
		ipScales	:	ITcVnContainer;	(* Container with the scaling parameters of each feature (type ContainerType_Vector_REAL or ContainerType_Vector_LREAL). *)
	END_VAR
	VAR_IN_OUT
		fInverseSample	:	REAL;	(* Returns the inversed sample. *)
	END_VAR
	VAR_INPUT
		fA	:	LREAL;	(* represents the lower bound of the range for TCVN_FST1_MINMAX *)
		fB	:	LREAL;	(* represents the upper bound of the range for TCVN_FST1_MINMAX *)
		hrPrev	:	HRESULT;	(* HRESULT indicating the result of previous operations (If SUCCEEDED(hrPrev) equals false, no operation is executed.) *)
	END_VAR

END_FUNCTION

// Functions/Machine Learning/F_VN_InverseFeatureTransform

	{attribute 'TcIecLibraryType'}
	{attribute 'external_name' := 'F_VN_InverseFeatureTransform_GUID_DDE5C7AA_8679_4435_FF7F_AB60919BDE1C'}
	(* Apply an inverse feature transform to one or more sample(s). *)
	FUNCTION F_VN_InverseFeatureTransform : HRESULT
	VAR_INPUT
		ipFeatureTransform	:	ITcVnMlModel;	(* Feature transform instance to be used *)
		ipSamples	:	ITcUnknown;	(* Container holding one or more of input sample(s) (ContainerType_Vector_REAL, ContainerType_Vector_LREAL, ContainerType_Vector_Vector_REAL, or ContainerType_Vector_Vector_LREAL) *)
		pipTransformed	:	POINTER TO ITcUnknown;	(* Returns the transformed sample(s) using the same type like ipSamples *)
		hrPrev	:	HRESULT;	(* HRESULT indicating the result of previous operations (If SUCCEEDED(hrPrev) equals false, no operation is executed.) *)
	END_VAR

END_FUNCTION

// Functions/Machine Learning/F_VN_PredictBatch

	{attribute 'TcIecLibraryType'}
	{attribute 'external_name' := 'F_VN_PredictBatch_GUID_96755CC6_5D1C_4EE3_D4A0_6FDB6D1103E4'}
	(* Compute predictions for a batch of samples. *)
	FUNCTION F_VN_PredictBatch : HRESULT
	VAR_INPUT
		ipMlModel	:	ITcVnMlModel;	(* Classifier or regressor to be used *)
		ipSamples	:	ITcUnknown;	(* Container holding a batch of input samples (ContainerType_Vector_Vector_REAL or ContainerType_Vector_Vector_LREAL) *)
		ipPredictions	:	REFERENCE TO ITcVnContainer;	(* Returns the predicted outputs (depending on ipSamples; class labels (for classification, ContainerType_Vector_DINT) or real-valued predictions (for regression with scalar output, ContainerType_Vector_REAL or ContainerType_Vector_LREAL; for regression with vectorial output, ContainerType_Vector_Vector_REAL or ContainerType_Vector_Vector_LREAL)) *)
		hrPrev	:	HRESULT;	(* HRESULT indicating the result of previous operations (If SUCCEEDED(hrPrev) equals false, no operation is executed.) *)
	END_VAR

END_FUNCTION

// Functions/Machine Learning/F_VN_PredictBatchExp

	{attribute 'TcIecLibraryType'}
	{attribute 'external_name' := 'F_VN_PredictBatchExp_GUID_2890470D_A1AE_4AFA_E1EC_B2208C6B1665'}
	(* Compute predictions for a batch of samples. (expert function) *)
	FUNCTION F_VN_PredictBatchExp : HRESULT
	VAR_INPUT
		ipMlModel	:	ITcVnMlModel;	(* Classifier or regressor to be used *)
		ipSamples	:	ITcUnknown;	(* Container holding a batch of input samples (ContainerType_Vector_Vector_REAL or ContainerType_Vector_Vector_LREAL) *)
		ipPredictions	:	REFERENCE TO ITcVnContainer;	(* Returns the predicted outputs (depending on ipSamples; class labels (for classification, ContainerType_Vector_DINT) or real-valued predictions (for regression with scalar output, ContainerType_Vector_REAL or ContainerType_Vector_LREAL; for regression with vectorial output, ContainerType_Vector_Vector_REAL or ContainerType_Vector_Vector_LREAL)) *)
		ipNovelties	:	REFERENCE TO ITcVnContainer;	(* Returns the degree of novelty (0.0 if a sample is completely known; > 0.0 otherwise) of each sample (ContainerType_Vector_REAL; optional, set to 0 if not required) *)
		hrPrev	:	HRESULT;	(* HRESULT indicating the result of previous operations (If SUCCEEDED(hrPrev) equals false, no operation is executed.) *)
	END_VAR

END_FUNCTION

// Functions/Machine Learning/F_VN_PredictSampleClass

	{attribute 'TcIecLibraryType'}
	{attribute 'external_name' := 'F_VN_PredictSampleClass_GUID_A502DF80_050A_4D3C_CB9F_AAC726B2AEA8'}
	(* Classify a single sample. *)
	FUNCTION F_VN_PredictSampleClass : HRESULT
	VAR_INPUT
		ipClassifier	:	ITcVnMlModel;	(* Classifier to be used *)
		ipSample	:	ITcUnknown;	(* Container holding a single input sample (ContainerType_Vector_REAL or ContainerType_Vector_LREAL) *)
	END_VAR
	VAR_IN_OUT
		nClass	:	DINT;	(* Returns the classification result *)
	END_VAR
	VAR_INPUT
		hrPrev	:	HRESULT;	(* HRESULT indicating the result of previous operations (If SUCCEEDED(hrPrev) equals false, no operation is executed.) *)
	END_VAR

END_FUNCTION

// Functions/Machine Learning/F_VN_PredictSampleClassExp

	{attribute 'TcIecLibraryType'}
	{attribute 'external_name' := 'F_VN_PredictSampleClassExp_GUID_91E76752_8554_46CC_F737_E24CAE2B2AA7'}
	(* Classify a single sample. (expert function) *)
	FUNCTION F_VN_PredictSampleClassExp : HRESULT
	VAR_INPUT
		ipClassifier	:	ITcVnMlModel;	(* Classifier to be used *)
		ipSample	:	ITcUnknown;	(* Container holding a single input sample (ContainerType_Vector_REAL or ContainerType_Vector_LREAL) *)
	END_VAR
	VAR_IN_OUT
		nClass	:	DINT;	(* Returns the classification result *)
	END_VAR
	VAR_INPUT
		fNovelty	:	REFERENCE TO REAL;	(* Returns the degree of novelty (0.0 if a sample is completely known; > 0.0 otherwise) of the presented sample (optional, set to 0 if not required) *)
		hrPrev	:	HRESULT;	(* HRESULT indicating the result of previous operations (If SUCCEEDED(hrPrev) equals false, no operation is executed.) *)
	END_VAR

END_FUNCTION

// Functions/Machine Learning/F_VN_PredictSampleScalar

	{attribute 'TcIecLibraryType'}
	{attribute 'external_name' := 'F_VN_PredictSampleScalar_GUID_4B79A184_9689_491B_F6F5_0C645E446AB0'}
	(* Compute a scalar prediction for a single sample. *)
	FUNCTION F_VN_PredictSampleScalar : HRESULT
	VAR_INPUT
		ipRegressor	:	ITcVnMlModel;	(* Regressor to be used *)
		ipSample	:	ITcUnknown;	(* Container holding a single input sample (ContainerType_Vector_REAL or ContainerType_Vector_LREAL) *)
	END_VAR
	VAR_IN_OUT
		fPrediction	:	REAL;	(* Returns the predicted output *)
	END_VAR
	VAR_INPUT
		hrPrev	:	HRESULT;	(* HRESULT indicating the result of previous operations (If SUCCEEDED(hrPrev) equals false, no operation is executed.) *)
	END_VAR

END_FUNCTION

// Functions/Machine Learning/F_VN_PredictSampleScalarExp

	{attribute 'TcIecLibraryType'}
	{attribute 'external_name' := 'F_VN_PredictSampleScalarExp_GUID_D90DCA93_8674_4052_D5F4_0C87FE32A90F'}
	(* Compute a scalar prediction for a single sample. (expert function) *)
	FUNCTION F_VN_PredictSampleScalarExp : HRESULT
	VAR_INPUT
		ipRegressor	:	ITcVnMlModel;	(* Regressor to be used *)
		ipSample	:	ITcUnknown;	(* Container holding a single input sample (ContainerType_Vector_REAL or ContainerType_Vector_LREAL) *)
	END_VAR
	VAR_IN_OUT
		fPrediction	:	REAL;	(* Returns the predicted output *)
	END_VAR
	VAR_INPUT
		fNovelty	:	REFERENCE TO REAL;	(* Returns the degree of novelty (0.0 if a sample is completely known; > 0.0 otherwise) of the presented sample (optional, set to 0 if not required) *)
		hrPrev	:	HRESULT;	(* HRESULT indicating the result of previous operations (If SUCCEEDED(hrPrev) equals false, no operation is executed.) *)
	END_VAR

END_FUNCTION

// Functions/Machine Learning/F_VN_PredictSampleVector

	{attribute 'TcIecLibraryType'}
	{attribute 'external_name' := 'F_VN_PredictSampleVector_GUID_F85E5A95_3D2F_4D0A_EBAF_E0CA4087A8C5'}
	(* Compute a vectorial prediction for a single sample. *)
	FUNCTION F_VN_PredictSampleVector : HRESULT
	VAR_INPUT
		ipRegressor	:	ITcVnMlModel;	(* Regressor to be used *)
		ipSample	:	ITcUnknown;	(* Container holding a single input sample (ContainerType_Vector_REAL or ContainerType_Vector_LREAL) *)
		ipPrediction	:	REFERENCE TO ITcVnContainer;	(* Returns the predicted output (ContainerType_Vector_REAL or ContainerType_Vector_LREAL, depending on ipSample) *)
		hrPrev	:	HRESULT;	(* HRESULT indicating the result of previous operations (If SUCCEEDED(hrPrev) equals false, no operation is executed.) *)
	END_VAR

END_FUNCTION

// Functions/Machine Learning/F_VN_PredictSampleVectorExp

	{attribute 'TcIecLibraryType'}
	{attribute 'external_name' := 'F_VN_PredictSampleVectorExp_GUID_E800AF60_8BA4_46F1_D73D_9D44C5E6162F'}
	(* Compute a vectorial prediction for a single sample. (expert function) *)
	FUNCTION F_VN_PredictSampleVectorExp : HRESULT
	VAR_INPUT
		ipRegressor	:	ITcVnMlModel;	(* Regressor to be used *)
		ipSample	:	ITcUnknown;	(* Container holding a single input sample (ContainerType_Vector_REAL or ContainerType_Vector_LREAL) *)
		ipPrediction	:	REFERENCE TO ITcVnContainer;	(* Returns the predicted output (ContainerType_Vector_REAL or ContainerType_Vector_LREAL, depending on ipSample) *)
		fNovelty	:	REFERENCE TO REAL;	(* Returns the degree of novelty (0.0 if a sample is completely known; > 0.0 otherwise) of the presented sample (optional, set to 0 if not required) *)
		hrPrev	:	HRESULT;	(* HRESULT indicating the result of previous operations (If SUCCEEDED(hrPrev) equals false, no operation is executed.) *)
	END_VAR

END_FUNCTION

// Functions/Machine Learning/F_VN_FeatureScaling

	{attribute 'TcIecLibraryType'}
	{attribute 'external_name' := 'F_VN_FeatureScaling_GUID_70C62B2C_EA2E_4B8B_CC3A_9A38E2BB0731'}
	(* Apply a feature scaling to one or more sample(s). *)
	FUNCTION F_VN_FeatureScaling : HRESULT
	VAR_INPUT
		ipSamples	:	ITcVnContainer;	(* Container holding one or more input sample(s) (ContainerType_Vector_REAL, ContainerType_Vector_LREAL, ContainerType_Vector_Vector_REAL, or ContainerType_Vector_Vector_LREAL) *)
		ipScales	:	ITcVnContainer;	(* Container with the scaling parameters of each feature (type ContainerType_Vector_REAL or ContainerType_Vector_LREAL). *)
		ipScaledSamples	:	REFERENCE TO ITcVnContainer;	(* Returns the scaled sample(s) using the same type like ipSamples. If the same container ipSamples is uesd, the source data will be replaced. *)
		hrPrev	:	HRESULT;	(* HRESULT indicating the result of previous operations (If SUCCEEDED(hrPrev) equals false, no operation is executed.) *)
	END_VAR

END_FUNCTION

// Functions/Machine Learning/F_VN_FeatureScalingExp

	{attribute 'TcIecLibraryType'}
	{attribute 'external_name' := 'F_VN_FeatureScalingExp_GUID_89C1B59C_5137_4504_E1FB_D61319B47D2D'}
	(* Apply a feature scaling to one or more sample(s) and get output range between [fA, fB] in the case of TCVN_FST1_MINMAX.  (expert function) *)
	FUNCTION F_VN_FeatureScalingExp : HRESULT
	VAR_INPUT
		ipSamples	:	ITcVnContainer;	(* Container holding one or more input sample(s) (ContainerType_Vector_REAL, ContainerType_Vector_LREAL, ContainerType_Vector_Vector_REAL, or ContainerType_Vector_Vector_LREAL) *)
		ipScales	:	ITcVnContainer;	(* Container with the scaling parameters of each feature (type ContainerType_Vector_REAL or ContainerType_Vector_LREAL). *)
		ipScaledSamples	:	REFERENCE TO ITcVnContainer;	(* Returns the scaled sample(s) using the same type like ipSamples. If the same container ipSamples is uesd, the source data will be replaced. *)
		fA	:	LREAL;	(* represents the lower bound of the range for TCVN_FST1_MINMAX *)
		fB	:	LREAL;	(* represents the upper bound of the range for TCVN_FST1_MINMAX *)
		hrPrev	:	HRESULT;	(* HRESULT indicating the result of previous operations (If SUCCEEDED(hrPrev) equals false, no operation is executed.) *)
	END_VAR

END_FUNCTION

// Functions/Machine Learning/F_VN_TrainBatch

	{attribute 'TcIecLibraryType'}
	{attribute 'external_name' := 'F_VN_TrainBatch_GUID_9C8BD443_B8CB_4423_D9E4_F16627402CD5'}
	(* Train a classifier, a clusterer, a novelty detector, or a regressor with a batch of samples. On-line trainable models are trained once with each sample. Depending on the application and the number of available training samples, repeated training of such models with the same data may improve the results. *)
	FUNCTION F_VN_TrainBatch : HRESULT
	VAR_INPUT
		ipMlModel	:	ITcVnMlModel;	(* Classifier, clusterer, novelty detector, or regressor to be used *)
		ipSamples	:	ITcUnknown;	(* Container holding a batch of input samples (ContainerType_Vector_Vector_REAL or ContainerType_Vector_Vector_LREAL) *)
		ipOutputs	:	ITcVnContainer;	(* Class labels (for classification, ContainerType_Vector_DINT) or target outputs (for regression with scalar output, ContainerType_Vector_REAL or ContainerType_Vector_LREAL; for regression with vectorial output, ContainerType_Vector_Vector_REAL or ContainerType_Vector_Vector_LREAL) to be learnt (must be 0 for clusterers and for novelty detectors) *)
		hrPrev	:	HRESULT;	(* HRESULT indicating the result of previous operations (If SUCCEEDED(hrPrev) equals false, no operation is executed.) *)
	END_VAR

END_FUNCTION

// Functions/Machine Learning/F_VN_TrainBatchClusters

	{attribute 'TcIecLibraryType'}
	{attribute 'external_name' := 'F_VN_TrainBatchClusters_GUID_C8592228_94CB_40E3_EA8C_49A9E7D25B68'}
	(* Train a clusterer with a batch of samples and return the IDs of the clusters the samples have been assigned to, if requested. On-line trainable clusterers are trained once with each sample. Depending on the application and the number of available training samples, repeated training of such models with the same data may improve the results. *)
	FUNCTION F_VN_TrainBatchClusters : HRESULT
	VAR_INPUT
		ipClusterer	:	ITcVnMlModel;	(* Clusterer to be used *)
		ipSamples	:	ITcUnknown;	(* Container holding a batch of input samples (ContainerType_Vector_Vector_REAL or ContainerType_Vector_Vector_LREAL) *)
		ipClusters	:	REFERENCE TO ITcVnContainer;	(* Returns the IDs of the clusters the samples have been assigned to (ContainerType_Vector_DINT; optional, set to 0 if not required) *)
		hrPrev	:	HRESULT;	(* HRESULT indicating the result of previous operations (If SUCCEEDED(hrPrev) equals false, no operation is executed.) *)
	END_VAR

END_FUNCTION

// Functions/Machine Learning/F_VN_TrainSample

	{attribute 'TcIecLibraryType'}
	{attribute 'external_name' := 'F_VN_TrainSample_GUID_80158E83_F794_44E9_E8E2_4B54C8B0B0DE'}
	(* Train a clusterer or a novelty detector with a single sample. *)
	FUNCTION F_VN_TrainSample : HRESULT
	VAR_INPUT
		ipMlModel	:	ITcVnMlModel;	(* Clusterer or novelty detector to be used *)
		ipSample	:	ITcUnknown;	(* Container holding a single input sample (ContainerType_Vector_REAL or ContainerType_Vector_LREAL) *)
		hrPrev	:	HRESULT;	(* HRESULT indicating the result of previous operations (If SUCCEEDED(hrPrev) equals false, no operation is executed.) *)
	END_VAR

END_FUNCTION

// Functions/Machine Learning/F_VN_TrainSampleClass

	{attribute 'TcIecLibraryType'}
	{attribute 'external_name' := 'F_VN_TrainSampleClass_GUID_EAD5B0F2_94FC_4598_EE5C_0D1D51C50E4C'}
	(* Train a classifier with a single sample. *)
	FUNCTION F_VN_TrainSampleClass : HRESULT
	VAR_INPUT
		ipClassifier	:	ITcVnMlModel;	(* Classifier to be used *)
		ipSample	:	ITcUnknown;	(* Container holding a single input sample (ContainerType_Vector_REAL or ContainerType_Vector_LREAL) *)
		nClass	:	DINT;	(* Class label to be learnt *)
		hrPrev	:	HRESULT;	(* HRESULT indicating the result of previous operations (If SUCCEEDED(hrPrev) equals false, no operation is executed.) *)
	END_VAR

END_FUNCTION

// Functions/Machine Learning/F_VN_TrainSampleCluster

	{attribute 'TcIecLibraryType'}
	{attribute 'external_name' := 'F_VN_TrainSampleCluster_GUID_DB4D9AA0_1F50_4112_E6E6_DF4AEF363E16'}
	(* Train a clusterer with a single sample and return the ID of the cluster the sample has been assigned to, if requested. The clusterer must be online trainable. *)
	FUNCTION F_VN_TrainSampleCluster : HRESULT
	VAR_INPUT
		ipClusterer	:	ITcVnMlModel;	(* Clusterer to be used *)
		ipSample	:	ITcUnknown;	(* Container holding a single input sample (ContainerType_Vector_REAL or ContainerType_Vector_LREAL) *)
		nCluster	:	REFERENCE TO DINT;	(* Returns the ID of the cluster the sample has been assigned to (If the pointer is 0, no cluster ID is requested.) *)
		hrPrev	:	HRESULT;	(* HRESULT indicating the result of previous operations (If SUCCEEDED(hrPrev) equals false, no operation is executed.) *)
	END_VAR

END_FUNCTION

// Functions/Machine Learning/F_VN_TrainSampleScalar

	{attribute 'TcIecLibraryType'}
	{attribute 'external_name' := 'F_VN_TrainSampleScalar_GUID_B3CEFCE7_41B6_4AC1_E4C4_3A349757906E'}
	(* Train a regressor with a single sample and scalar output. *)
	FUNCTION F_VN_TrainSampleScalar : HRESULT
	VAR_INPUT
		ipRegressor	:	ITcVnMlModel;	(* Regressor to be used *)
		ipSample	:	ITcUnknown;	(* Container holding a single input sample (ContainerType_Vector_REAL or ContainerType_Vector_LREAL) *)
		fOutput	:	REAL;	(* Scalar output to be learnt *)
		hrPrev	:	HRESULT;	(* HRESULT indicating the result of previous operations (If SUCCEEDED(hrPrev) equals false, no operation is executed.) *)
	END_VAR

END_FUNCTION

// Functions/Machine Learning/F_VN_TrainSampleVector

	{attribute 'TcIecLibraryType'}
	{attribute 'external_name' := 'F_VN_TrainSampleVector_GUID_4A95B0BE_6C32_41F8_E952_35DEBF9CAB25'}
	(* Train a regressor with a single sample and vectorial output. *)
	FUNCTION F_VN_TrainSampleVector : HRESULT
	VAR_INPUT
		ipRegressor	:	ITcVnMlModel;	(* Regressor to be used *)
		ipSample	:	ITcUnknown;	(* Container holding a single input sample (ContainerType_Vector_REAL or ContainerType_Vector_LREAL) *)
		ipOutput	:	ITcVnContainer;	(* Vectorial output to be learnt (ContainerType_Vector_REAL or ContainerType_Vector_LREAL) *)
		hrPrev	:	HRESULT;	(* HRESULT indicating the result of previous operations (If SUCCEEDED(hrPrev) equals false, no operation is executed.) *)
	END_VAR

END_FUNCTION

// Functions/Drawing/F_VN_DrawArrow

	{attribute 'TcIecLibraryType'}
	{attribute 'external_name' := 'F_VN_DrawArrow_GUID_CEEC543B_81C4_4033_D7EC_7A437BB7DD12'}
	(* Draw an arrowed line. *)
	FUNCTION F_VN_DrawArrow : HRESULT
	VAR_INPUT
		nX1	:	UDINT;	(* x coordinate of the start point *)
		nY1	:	UDINT;	(* y coordinate of the start point *)
		nX2	:	UDINT;	(* x coordinate of the end point *)
		nY2	:	UDINT;	(* y coordinate of the end point *)
		ipDestImage	:	ITcVnImage;	(* Destination image *)
	END_VAR
	VAR_IN_OUT
		aColor	:	TcVnVector4_LREAL;	(* Color *)
	END_VAR
	VAR_INPUT
		nThickness	:	DINT;	(* Line thickness *)
		bDoubleHead	:	BOOL;	(* To draw an arrow on each side of the line. *)
		hrPrev	:	HRESULT;	(* HRESULT indicating the result of previous operations (If SUCCEEDED(hrPrev) equals false, no operation is executed.) *)
	END_VAR

END_FUNCTION

// Functions/Drawing/F_VN_DrawArrow_TcVnVector4_DINT

	{attribute 'TcIecLibraryType'}
	{attribute 'external_name' := 'F_VN_DrawArrow_TcVnVector4_DINT_GUID_22E4BE31_FB82_4A2F_ECB6_B93D963F9A70'}
	(* Draw an arrowed line. *)
	FUNCTION F_VN_DrawArrow_TcVnVector4_DINT : HRESULT
	VAR_IN_OUT
		aLine	:	TcVnVector4_DINT;	(* The start and end point of a line segment [x1, y1, x2, y2] *)
	END_VAR
	VAR_INPUT
		ipDestImage	:	ITcVnImage;	(* Destination image *)
	END_VAR
	VAR_IN_OUT
		aColor	:	TcVnVector4_LREAL;	(* Color *)
	END_VAR
	VAR_INPUT
		nThickness	:	DINT;	(* Line thickness *)
		bDoubleHead	:	BOOL;	(* To draw an arrow on each side of the line. *)
		hrPrev	:	HRESULT;	(* HRESULT indicating the result of previous operations (If SUCCEEDED(hrPrev) equals false, no operation is executed.) *)
	END_VAR

END_FUNCTION

// Functions/Drawing/F_VN_DrawArrowExp

	{attribute 'TcIecLibraryType'}
	{attribute 'external_name' := 'F_VN_DrawArrowExp_GUID_770711B5_5C2A_4A39_F178_B6656D90D5DF'}
	(* Draws an arrowed line. (expert function) *)
	FUNCTION F_VN_DrawArrowExp : HRESULT
	VAR_INPUT
		nX1	:	UDINT;	(* x coordinate of the start point *)
		nY1	:	UDINT;	(* y coordinate of the start point *)
		nX2	:	UDINT;	(* x coordinate of the end point *)
		nY2	:	UDINT;	(* y coordinate of the end point *)
		ipDestImage	:	ITcVnImage;	(* Destination image *)
	END_VAR
	VAR_IN_OUT
		aColor	:	TcVnVector4_LREAL;	(* Color *)
	END_VAR
	VAR_INPUT
		nThickness	:	DINT;	(* Line thickness *)
		bDoubleHead	:	BOOL;	(* To draw an arrow on each side of the line. *)
		eLineType	:	ETcVnLineType;	(* Line type *)
		nShift	:	UDINT;	(* Fractional bits of the coordinates (bit shift) *)
		fTipLenght	:	LREAL;	(* Lenght of the arrow's tip as a fraction of the line's lenght *)
		hrPrev	:	HRESULT;	(* HRESULT indicating the result of previous operations (If SUCCEEDED(hrPrev) equals false, no operation is executed.) *)
	END_VAR

END_FUNCTION

// Functions/Drawing/F_VN_DrawArrowExp_TcVnVector4_DINT

	{attribute 'TcIecLibraryType'}
	{attribute 'external_name' := 'F_VN_DrawArrowExp_TcVnVector4_DINT_GUID_046CAD01_98B8_447D_E9D2_B90F2D0C6441'}
	(* Draws an arrowed line. (expert function) *)
	FUNCTION F_VN_DrawArrowExp_TcVnVector4_DINT : HRESULT
	VAR_IN_OUT
		aLine	:	TcVnVector4_DINT;	(* The start and end point of a line segment [x1, y1, x2, y2] *)
	END_VAR
	VAR_INPUT
		ipDestImage	:	ITcVnImage;	(* Destination image *)
	END_VAR
	VAR_IN_OUT
		aColor	:	TcVnVector4_LREAL;	(* Color *)
	END_VAR
	VAR_INPUT
		nThickness	:	DINT;	(* Line thickness *)
		bDoubleHead	:	BOOL;	(* To draw an arrow on each side of the line. *)
		eLineType	:	ETcVnLineType;	(* Line type *)
		nShift	:	UDINT;	(* Fractional bits of the coordinates (bit shift) *)
		fTipLenght	:	LREAL;	(* Lenght of the arrow's tip as a fraction of the line's lenght *)
		hrPrev	:	HRESULT;	(* HRESULT indicating the result of previous operations (If SUCCEEDED(hrPrev) equals false, no operation is executed.) *)
	END_VAR

END_FUNCTION

// Functions/Drawing/F_VN_DrawCircle

	{attribute 'TcIecLibraryType'}
	{attribute 'external_name' := 'F_VN_DrawCircle_GUID_0A3D0612_E45C_4DC6_DF0F_3C05A1336793'}
	(* Draws a circle. *)
	FUNCTION F_VN_DrawCircle : HRESULT
	VAR_INPUT
		nCenterX	:	UDINT;	(* x coordinate of the center *)
		nCenterY	:	UDINT;	(* y coordinate of the center *)
		nRadius	:	UDINT;	(* Radius *)
		ipDestImage	:	ITcVnImage;	(* Destination image *)
	END_VAR
	VAR_IN_OUT
		aColor	:	TcVnVector4_LREAL;	(* Color *)
	END_VAR
	VAR_INPUT
		nThickness	:	DINT;	(* Line thickness (if negative, the circle is filled) *)
		hrPrev	:	HRESULT;	(* HRESULT indicating the result of previous operations (If SUCCEEDED(hrPrev) equals false, no operation is executed.) *)
	END_VAR

END_FUNCTION

// Functions/Drawing/F_VN_DrawCircleExp

	{attribute 'TcIecLibraryType'}
	{attribute 'external_name' := 'F_VN_DrawCircleExp_GUID_04823D91_CA81_4762_F55B_FC13AFFFE224'}
	(* Draws a circle. *)
	FUNCTION F_VN_DrawCircleExp : HRESULT
	VAR_INPUT
		nCenterX	:	UDINT;	(* x coordinate of the center *)
		nCenterY	:	UDINT;	(* y coordinate of the center *)
		nRadius	:	UDINT;	(* Radius *)
		ipDestImage	:	ITcVnImage;	(* Destination image *)
	END_VAR
	VAR_IN_OUT
		aColor	:	TcVnVector4_LREAL;	(* Color *)
	END_VAR
	VAR_INPUT
		nThickness	:	DINT;	(* Line thickness (if negative, the circle is filled) *)
		eLineType	:	ETcVnLineType;	(* Line type *)
		hrPrev	:	HRESULT;	(* HRESULT indicating the result of previous operations (If SUCCEEDED(hrPrev) equals false, no operation is executed.) *)
	END_VAR

END_FUNCTION

// Functions/Drawing/F_VN_DrawCircles

	{attribute 'TcIecLibraryType'}
	{attribute 'external_name' := 'F_VN_DrawCircles_GUID_FC990D3E_7169_4842_DB60_1CCA83A20B8A'}
	(* Draws circles. *)
	FUNCTION F_VN_DrawCircles : HRESULT
	VAR_INPUT
		ipCircles	:	ITcVnContainer;	(* Container with circles (ContainerType_Vector_TcVnVector3_REAL; Each container element contains the x coordinate of the circle center [0], the y coordinate of the circle center [1], and the radius [2].) *)
		nCircleIndex	:	DINT;	(* Index of a specific circle to be drawn (if negative, all circles within the container are drawn) *)
		ipDestImage	:	ITcVnImage;	(* Destination image *)
	END_VAR
	VAR_IN_OUT
		aColor	:	TcVnVector4_LREAL;	(* Color *)
	END_VAR
	VAR_INPUT
		nThickness	:	DINT;	(* Line thickness (if negative, the circle is filled) *)
		hrPrev	:	HRESULT;	(* HRESULT indicating the result of previous operations (If SUCCEEDED(hrPrev) equals false, no operation is executed.) *)
	END_VAR

END_FUNCTION

// Functions/Drawing/F_VN_DrawCirclesExp

	{attribute 'TcIecLibraryType'}
	{attribute 'external_name' := 'F_VN_DrawCirclesExp_GUID_AFF73A37_6F22_4B41_DEC5_C85A0CA1A59C'}
	(* Draws circles. (expert function) *)
	FUNCTION F_VN_DrawCirclesExp : HRESULT
	VAR_INPUT
		ipCircles	:	ITcVnContainer;	(* Container with circles (ContainerType_Vector_TcVnVector3_REAL; Each container element contains the x coordinate of the circle center [0], the y coordinate of the circle center [1], and the radius [2].) *)
		nCircleIndex	:	DINT;	(* Index of a specific circle to be drawn (if negative, all circles within the container are drawn) *)
		ipDestImage	:	ITcVnImage;	(* Destination image *)
	END_VAR
	VAR_IN_OUT
		aColor	:	TcVnVector4_LREAL;	(* Color *)
	END_VAR
	VAR_INPUT
		nThickness	:	DINT;	(* Line thickness (if negative, the circle is filled) *)
		eLineType	:	ETcVnLineType;	(* Line type *)
		hrPrev	:	HRESULT;	(* HRESULT indicating the result of previous operations (If SUCCEEDED(hrPrev) equals false, no operation is executed.) *)
	END_VAR

END_FUNCTION

// Functions/Drawing/F_VN_DrawCircularArc

	{attribute 'TcIecLibraryType'}
	{attribute 'external_name' := 'F_VN_DrawCircularArc_GUID_0D29C983_52AD_4911_CE04_F65ED67C5221'}
	(* Draws a circular arc. *)
	FUNCTION F_VN_DrawCircularArc : HRESULT
	VAR_IN_OUT
		stCircularArc	:	TcVnCircularArc;	(* Circular arc definition *)
	END_VAR
	VAR_INPUT
		ipDestImage	:	ITcVnImage;	(* Destination image *)
	END_VAR
	VAR_IN_OUT
		aColor	:	TcVnVector4_LREAL;	(* Color *)
	END_VAR
	VAR_INPUT
		nThickness	:	DINT;	(* Line thickness (if negative, the arc is filled) *)
		hrPrev	:	HRESULT;	(* HRESULT indicating the result of previous operations (If SUCCEEDED(hrPrev) equals false, no operation is executed.) *)
	END_VAR

END_FUNCTION

// Functions/Drawing/F_VN_DrawCircularArcExp

	{attribute 'TcIecLibraryType'}
	{attribute 'external_name' := 'F_VN_DrawCircularArcExp_GUID_36C082D0_7BE2_445B_D2B6_BA82ED2256EF'}
	(* Draws a circular arc. (expert function) *)
	FUNCTION F_VN_DrawCircularArcExp : HRESULT
	VAR_IN_OUT
		stCircularArc	:	TcVnCircularArc;	(* Circular arc definition *)
	END_VAR
	VAR_INPUT
		ipDestImage	:	ITcVnImage;	(* Destination image *)
	END_VAR
	VAR_IN_OUT
		aColor	:	TcVnVector4_LREAL;	(* Color *)
	END_VAR
	VAR_INPUT
		nThickness	:	DINT;	(* Line thickness (if negative, the arc is filled) *)
		eLineType	:	ETcVnLineType;	(* Line type *)
		hrPrev	:	HRESULT;	(* HRESULT indicating the result of previous operations (If SUCCEEDED(hrPrev) equals false, no operation is executed.) *)
	END_VAR

END_FUNCTION

// Functions/Drawing/F_VN_DrawComponents

	{attribute 'TcIecLibraryType'}
	{attribute 'external_name' := 'F_VN_DrawComponents_GUID_06E1DAFB_7E1B_45FB_CBE9_472D937E824E'}
	(* Draw the results of connected component function. *)
	FUNCTION F_VN_DrawComponents : HRESULT
	VAR_INPUT
		ipLabelImage	:	ITcVnImage;	(* Image contains labels for each pixel (1 channel DINT or UINT). *)
		nLabelID	:	DINT;	(* Value of a specific label to be drawn (if negative, all components within the image are drawn) *)
		ipDestImage	:	REFERENCE TO ITcVnImage;	(* Destination image (An appropriate image will be created if required. The output image is 1 or 3 channels USINT). *)
		bShowLabelID	:	BOOL;	(* Show label ID in the center of the component on the destination image *)
		hrPrev	:	HRESULT;	(* HRESULT indicating the result of previous operations (If SUCCEEDED(hrPrev) equals false, no operation is executed.) *)
	END_VAR

END_FUNCTION

// Functions/Drawing/F_VN_DrawComponentsExp

	{attribute 'TcIecLibraryType'}
	{attribute 'external_name' := 'F_VN_DrawComponentsExp_GUID_88845F55_AD67_4D75_C46B_48444CE1EC3B'}
	(* Draw the results of connected component function. (expert function) *)
	FUNCTION F_VN_DrawComponentsExp : HRESULT
	VAR_INPUT
		ipLabelImage	:	ITcVnImage;	(* Image contains labels for each pixel (1 channel DINT or UINT). *)
		nLabelID	:	DINT;	(* Value of a specific label to be drawn (if negative, all components within the image are drawn) *)
		ipDestImage	:	REFERENCE TO ITcVnImage;	(* Destination image (An appropriate image will be created if required. The output image is 1 or 3 channels USINT). *)
		bShowLabelID	:	BOOL;	(* Show lable ID in the center of the component on the destination image *)
	END_VAR
	VAR_IN_OUT
		aColor	:	TcVnVector4_LREAL;	(* Color to draw the components (for {-1, -1, -1, -1}, a random color is chosen for each component) *)
	END_VAR
	VAR_INPUT
		nThickness	:	DINT;	(* Text line thickness *)
		fFontScale	:	LREAL;	(* Scaling factor for the text *)
		hrPrev	:	HRESULT;	(* HRESULT indicating the result of previous operations (If SUCCEEDED(hrPrev) equals false, no operation is executed.) *)
	END_VAR

END_FUNCTION

// Functions/Drawing/F_VN_DrawContours

	{attribute 'TcIecLibraryType'}
	{attribute 'external_name' := 'F_VN_DrawContours_GUID_52E55E83_C98B_490B_CF6C_260DF3AB8539'}
	(* Draws a single point set or multiple point sets that are interpreted as contours. *)
	FUNCTION F_VN_DrawContours : HRESULT
	VAR_INPUT
		ipContours	:	ITcVnContainer;	(* Single contour (ContainerType_Vector_TcVnPoint2_DINT) or multiple contours (ContainerType_Vector_Vector_TcVnPoint2_DINT) *)
		nContourIndex	:	DINT;	(* Index of a specific contour to be drawn (if negative, all contours within the container are drawn) *)
		ipDestImage	:	ITcVnImage;	(* Destination image *)
	END_VAR
	VAR_IN_OUT
		aColor	:	TcVnVector4_LREAL;	(* Color *)
	END_VAR
	VAR_INPUT
		nThickness	:	DINT;	(* Line thickness (if negative, the contours are filled) *)
		hrPrev	:	HRESULT;	(* HRESULT indicating the result of previous operations (If SUCCEEDED(hrPrev) equals false, no operation is executed.) *)
	END_VAR

END_FUNCTION

// Functions/Drawing/F_VN_DrawContoursExp

	{attribute 'TcIecLibraryType'}
	{attribute 'external_name' := 'F_VN_DrawContoursExp_GUID_21880E46_7ACA_4DE9_D3F9_A110CB83A9E1'}
	(* Draws a single point set or multiple point sets that are interpreted as contours. (expert function) *)
	FUNCTION F_VN_DrawContoursExp : HRESULT
	VAR_INPUT
		ipContours	:	ITcVnContainer;	(* Single contour (ContainerType_Vector_TcVnPoint2_DINT) or multiple contours (ContainerType_Vector_Vector_TcVnPoint2_DINT) *)
		nContourIndex	:	DINT;	(* Index of a specific contour to be drawn (if negative, all contours within the container are drawn) *)
		ipDestImage	:	ITcVnImage;	(* Destination image *)
	END_VAR
	VAR_IN_OUT
		aColor	:	TcVnVector4_LREAL;	(* Color *)
	END_VAR
	VAR_INPUT
		nThickness	:	DINT;	(* Line thickness (if negative, the contours are filled) *)
		eLineType	:	ETcVnLineType;	(* Line type *)
		ipHierarchy	:	ITcVnContainer;	(* Contour hierarchy (ContainerType_Vector_TcVnVector4_DINT) *)
		nMaxLevel	:	DINT;	(* Maximum level of contours to be drawn *)
	END_VAR
	VAR_IN_OUT
		aOffset	:	TcVnPoint;	(* Offset by which every contour point is shifted *)
	END_VAR
	VAR_INPUT
		hrPrev	:	HRESULT;	(* HRESULT indicating the result of previous operations (If SUCCEEDED(hrPrev) equals false, no operation is executed.) *)
	END_VAR

END_FUNCTION

// Functions/Drawing/F_VN_DrawEllipse

	{attribute 'TcIecLibraryType'}
	{attribute 'external_name' := 'F_VN_DrawEllipse_GUID_DBF8F0C4_4C67_46CE_D848_C58FBC7DD56B'}
	(* Draws an ellipse. *)
	FUNCTION F_VN_DrawEllipse : HRESULT
	VAR_IN_OUT
		stEllipse	:	TcVnRotatedRectangle;	(* Ellipse to be drawn (rotation angle in degrees) *)
	END_VAR
	VAR_INPUT
		ipDestImage	:	ITcVnImage;	(* Destination image *)
	END_VAR
	VAR_IN_OUT
		aColor	:	TcVnVector4_LREAL;	(* Color *)
	END_VAR
	VAR_INPUT
		nThickness	:	DINT;	(* Line thickness (if negative, the ellipse is filled) *)
		hrPrev	:	HRESULT;	(* HRESULT indicating the result of previous operations (If SUCCEEDED(hrPrev) equals false, no operation is executed.) *)
	END_VAR

END_FUNCTION

// Functions/Drawing/F_VN_DrawEllipseExp

	{attribute 'TcIecLibraryType'}
	{attribute 'external_name' := 'F_VN_DrawEllipseExp_GUID_2AF46088_8E51_40A6_FE7F_9BC3E57CBEBB'}
	(* Draws an ellipse. (expert function) *)
	FUNCTION F_VN_DrawEllipseExp : HRESULT
	VAR_IN_OUT
		stEllipse	:	TcVnRotatedRectangle;	(* Ellipse to be drawn (rotation angle in degrees) *)
	END_VAR
	VAR_INPUT
		ipDestImage	:	ITcVnImage;	(* Destination image *)
	END_VAR
	VAR_IN_OUT
		aColor	:	TcVnVector4_LREAL;	(* Color *)
	END_VAR
	VAR_INPUT
		nThickness	:	DINT;	(* Line thickness (if negative, the ellipse is filled) *)
		eLineType	:	ETcVnLineType;	(* Line type *)
		hrPrev	:	HRESULT;	(* HRESULT indicating the result of previous operations (If SUCCEEDED(hrPrev) equals false, no operation is executed.) *)
	END_VAR

END_FUNCTION

// Functions/Drawing/F_VN_DrawKeypoints

	{attribute 'TcIecLibraryType'}
	{attribute 'external_name' := 'F_VN_DrawKeypoints_GUID_93ABBDB1_8042_42D3_D0FA_66BFBB1A7595'}
	(* Draws the keypoints for visualization purpose. *)
	FUNCTION F_VN_DrawKeypoints : HRESULT
	VAR_INPUT
		ipSrcImage	:	ITcVnImage;	(* Source image (elements of type USINT) *)
		ipKeyPoints	:	ITcVnContainer;	(* Container with the keypoints (ContainerType_Vector_TcVnKeyPoint) *)
		ipDestImage	:	REFERENCE TO ITcVnImage;	(* Destination image (An appropriate color image will be created if required.) *)
		hrPrev	:	HRESULT;	(* HRESULT indicating the result of previous operations (If SUCCEEDED(hrPrev) equals false, no operation is executed.) *)
	END_VAR

END_FUNCTION

// Functions/Drawing/F_VN_DrawKeypointsExp

	{attribute 'TcIecLibraryType'}
	{attribute 'external_name' := 'F_VN_DrawKeypointsExp_GUID_3D8030DF_36E8_4210_ED0A_BE074DBADE02'}
	(* Draws the keypoints for visualization purpose. (expert function) *)
	FUNCTION F_VN_DrawKeypointsExp : HRESULT
	VAR_INPUT
		ipSrcImage	:	ITcVnImage;	(* Source image (elements of type USINT) *)
		ipKeyPoints	:	ITcVnContainer;	(* Container with the keypoints (ContainerType_Vector_TcVnKeyPoint) *)
		ipDestImage	:	REFERENCE TO ITcVnImage;	(* Destination image (An appropriate color image will be created if required.) *)
	END_VAR
	VAR_IN_OUT
		aColor	:	TcVnVector4_LREAL;	(* Color to draw the keypoints (for {-1, -1, -1, -1}, a random color is chosen for each point) *)
	END_VAR
	VAR_INPUT
		eFlags	:	ETcVnDrawMatchesFlags;	(* A combination of flags to support overdrawing an existing destination image and/or drawing additional (Rich-)Keypoint information (size and orientation) *)
		hrPrev	:	HRESULT;	(* HRESULT indicating the result of previous operations (If SUCCEEDED(hrPrev) equals false, no operation is executed.) *)
	END_VAR

END_FUNCTION

// Functions/Drawing/F_VN_DrawLine

	{attribute 'TcIecLibraryType'}
	{attribute 'external_name' := 'F_VN_DrawLine_GUID_ED03D868_4B19_4819_EB99_FBA640562F9D'}
	(* Draws a line. *)
	FUNCTION F_VN_DrawLine : HRESULT
	VAR_INPUT
		nX1	:	UDINT;	(* x coordinate of the start point *)
		nY1	:	UDINT;	(* y coordinate of the start point *)
		nX2	:	UDINT;	(* x coordinate of the end point *)
		nY2	:	UDINT;	(* y coordinate of the end point *)
		ipDestImage	:	ITcVnImage;	(* Destination image *)
	END_VAR
	VAR_IN_OUT
		aColor	:	TcVnVector4_LREAL;	(* Color *)
	END_VAR
	VAR_INPUT
		nThickness	:	DINT;	(* Line thickness *)
		hrPrev	:	HRESULT;	(* HRESULT indicating the result of previous operations (If SUCCEEDED(hrPrev) equals false, no operation is executed.) *)
	END_VAR

END_FUNCTION

// Functions/Drawing/F_VN_DrawLineExp

	{attribute 'TcIecLibraryType'}
	{attribute 'external_name' := 'F_VN_DrawLineExp_GUID_B5539F8A_6270_4B3A_C60A_EC37BBCAA506'}
	(* Draws a line. (expert function) *)
	FUNCTION F_VN_DrawLineExp : HRESULT
	VAR_INPUT
		nX1	:	UDINT;	(* x coordinate of the start point *)
		nY1	:	UDINT;	(* y coordinate of the start point *)
		nX2	:	UDINT;	(* x coordinate of the end point *)
		nY2	:	UDINT;	(* y coordinate of the end point *)
		ipDestImage	:	ITcVnImage;	(* Destination image *)
	END_VAR
	VAR_IN_OUT
		aColor	:	TcVnVector4_LREAL;	(* Color *)
	END_VAR
	VAR_INPUT
		nThickness	:	DINT;	(* Line thickness *)
		eLineType	:	ETcVnLineType;	(* Line type *)
		nShift	:	UDINT;	(* Fractional bits of the coordinates (bit shift) *)
		hrPrev	:	HRESULT;	(* HRESULT indicating the result of previous operations (If SUCCEEDED(hrPrev) equals false, no operation is executed.) *)
	END_VAR

END_FUNCTION

// Functions/Drawing/F_VN_DrawLine_TcVnVector4_DINT

	{attribute 'TcIecLibraryType'}
	{attribute 'external_name' := 'F_VN_DrawLine_TcVnVector4_DINT_GUID_635925B3_EBAA_4B0D_EABD_843E4348CDFD'}
	(* Draws a line. *)
	FUNCTION F_VN_DrawLine_TcVnVector4_DINT : HRESULT
	VAR_IN_OUT
		aLine	:	TcVnVector4_DINT;	(* The start and end point of a line segment [x1, y1, x2, y2] *)
	END_VAR
	VAR_INPUT
		ipDestImage	:	ITcVnImage;	(* Destination image *)
	END_VAR
	VAR_IN_OUT
		aColor	:	TcVnVector4_LREAL;	(* Color *)
	END_VAR
	VAR_INPUT
		nThickness	:	DINT;	(* Line thickness *)
		hrPrev	:	HRESULT;	(* HRESULT indicating the result of previous operations (If SUCCEEDED(hrPrev) equals false, no operation is executed.) *)
	END_VAR

END_FUNCTION

// Functions/Drawing/F_VN_DrawLineExp_TcVnVector4_DINT

	{attribute 'TcIecLibraryType'}
	{attribute 'external_name' := 'F_VN_DrawLineExp_TcVnVector4_DINT_GUID_0337789F_0EF0_4341_E684_88149F0E9AFB'}
	(* Draws a line. (expert function) *)
	FUNCTION F_VN_DrawLineExp_TcVnVector4_DINT : HRESULT
	VAR_IN_OUT
		aLine	:	TcVnVector4_DINT;	(* The start and end point of a line segment [x1, y1, x2, y2] *)
	END_VAR
	VAR_INPUT
		ipDestImage	:	ITcVnImage;	(* Destination image *)
	END_VAR
	VAR_IN_OUT
		aColor	:	TcVnVector4_LREAL;	(* Color *)
	END_VAR
	VAR_INPUT
		nThickness	:	DINT;	(* Line thickness *)
		eLineType	:	ETcVnLineType;	(* Line type *)
		nShift	:	UDINT;	(* Fractional bits of the coordinates (bit shift) *)
		hrPrev	:	HRESULT;	(* HRESULT indicating the result of previous operations (If SUCCEEDED(hrPrev) equals false, no operation is executed.) *)
	END_VAR

END_FUNCTION

// Functions/Drawing/F_VN_DrawLine_TcVnVector4_LREAL

	{attribute 'TcIecLibraryType'}
	{attribute 'external_name' := 'F_VN_DrawLine_TcVnVector4_LREAL_GUID_98876D4F_6CE2_42CB_D1B5_7072A5879118'}
	(* Draws a line. *)
	FUNCTION F_VN_DrawLine_TcVnVector4_LREAL : HRESULT
	VAR_IN_OUT
		aLine	:	TcVnVector4_LREAL;	(* The first and second element describe the x and y component of the direction vector. The third and fourth element describe the x and y component of the position vector. *)
	END_VAR
	VAR_INPUT
		ipDestImage	:	ITcVnImage;	(* Destination image *)
	END_VAR
	VAR_IN_OUT
		aColor	:	TcVnVector4_LREAL;	(* Color *)
	END_VAR
	VAR_INPUT
		nThickness	:	DINT;	(* Line thickness *)
		hrPrev	:	HRESULT;	(* HRESULT indicating the result of previous operations (If SUCCEEDED(hrPrev) equals false, no operation is executed.) *)
	END_VAR

END_FUNCTION

// Functions/Drawing/F_VN_DrawLineExp_TcVnVector4_LREAL

	{attribute 'TcIecLibraryType'}
	{attribute 'external_name' := 'F_VN_DrawLineExp_TcVnVector4_LREAL_GUID_21EE7A8E_9F0D_43FD_D2FC_B4906DB3CA15'}
	(* Draws a line. (expert function) *)
	FUNCTION F_VN_DrawLineExp_TcVnVector4_LREAL : HRESULT
	VAR_IN_OUT
		aLine	:	TcVnVector4_LREAL;	(* The first and second element describe the x and y component of the direction vector. The third and fourth element describe the x and y component of the position vector. *)
	END_VAR
	VAR_INPUT
		ipDestImage	:	ITcVnImage;	(* Destination image *)
	END_VAR
	VAR_IN_OUT
		aColor	:	TcVnVector4_LREAL;	(* Color *)
	END_VAR
	VAR_INPUT
		nThickness	:	DINT;	(* Line thickness *)
		eLineType	:	ETcVnLineType;	(* Line type *)
		nShift	:	UDINT;	(* Fractional bits of the coordinates (bit shift) *)
		hrPrev	:	HRESULT;	(* HRESULT indicating the result of previous operations (If SUCCEEDED(hrPrev) equals false, no operation is executed.) *)
	END_VAR

END_FUNCTION

// Functions/Drawing/F_VN_DrawLines

	{attribute 'TcIecLibraryType'}
	{attribute 'external_name' := 'F_VN_DrawLines_GUID_1764AE9B_B2FD_4332_D4CC_9FE44EA7A930'}
	(* Draws lines. *)
	FUNCTION F_VN_DrawLines : HRESULT
	VAR_INPUT
		ipLines	:	ITcVnContainer;	(* Container with line descriptions (ContainerType_Vector_TcVnVector2_REAL: the distance from the origin [0] in pixels and the rotation angle [1] in radians. ContainerType_Vector_TcVnVector4_LREAL: the first and second element describe the x and y component of a vector collinear to the line. The third and fourth element describe the x and y component of a point on the line. ContainerType_Vector_TcVnVector4_DINT: start and end point [x1, y1, x2, y2]) *)
		nLineIndex	:	DINT;	(* Index of a specific line to be drawn (if negative, all lines within the container are drawn) *)
		ipDestImage	:	ITcVnImage;	(* Destination image *)
	END_VAR
	VAR_IN_OUT
		aColor	:	TcVnVector4_LREAL;	(* Color *)
	END_VAR
	VAR_INPUT
		nThickness	:	DINT;	(* Line thickness *)
		hrPrev	:	HRESULT;	(* HRESULT indicating the result of previous operations (If SUCCEEDED(hrPrev) equals false, no operation is executed.) *)
	END_VAR

END_FUNCTION

// Functions/Drawing/F_VN_DrawLinesExp

	{attribute 'TcIecLibraryType'}
	{attribute 'external_name' := 'F_VN_DrawLinesExp_GUID_2C770E40_ED43_4265_C4BD_103D074E2202'}
	(* Draws lines. (expert function) *)
	FUNCTION F_VN_DrawLinesExp : HRESULT
	VAR_INPUT
		ipLines	:	ITcVnContainer;	(* Container with line descriptions (ContainerType_Vector_TcVnVector2_REAL: the distance from the origin [0] in pixels and the rotation angle [1] in radians. ContainerType_Vector_TcVnVector4_LREAL: the first and second element describe the x and y component of a vector collinear to the line. The third and fourth element describe the x and y component of a point on the line. ContainerType_Vector_TcVnVector4_DINT: start and end point [x1, y1, x2, y2]) *)
		nLineIndex	:	DINT;	(* Index of a specific line to be drawn (if negative, all lines within the container are drawn) *)
		ipDestImage	:	ITcVnImage;	(* Destination image *)
	END_VAR
	VAR_IN_OUT
		aColor	:	TcVnVector4_LREAL;	(* Color *)
	END_VAR
	VAR_INPUT
		nThickness	:	DINT;	(* Line thickness *)
		eLineType	:	ETcVnLineType;	(* Line type *)
		nShift	:	UDINT;	(* Fractional bits of the coordinates (bit shift) *)
		hrPrev	:	HRESULT;	(* HRESULT indicating the result of previous operations (If SUCCEEDED(hrPrev) equals false, no operation is executed.) *)
	END_VAR

END_FUNCTION

// Functions/Drawing/F_VN_DrawMatches

	{attribute 'TcIecLibraryType'}
	{attribute 'external_name' := 'F_VN_DrawMatches_GUID_FCB983DC_0C19_42AF_FE28_ADB61B550CCA'}
	(* Draws the keypoints and matches for visualization purpose. *)
	FUNCTION F_VN_DrawMatches : HRESULT
	VAR_INPUT
		ipSrcImage1	:	ITcVnImage;	(* Source image 1 (elements of type USINT) *)
		ipKeyPoints1	:	ITcVnContainer;	(* Container with the keypoints 1 (ContainerType_Vector_TcVnKeyPoint) *)
		ipSrcImage2	:	ITcVnImage;	(* Source image 2 (elements of type USINT, must have the same number of channels as ipSrcImage1) *)
		ipKeyPoints2	:	ITcVnContainer;	(* Container with the keypoints 2 (ContainerType_Vector_TcVnKeyPoint) *)
		ipMatches1To2	:	ITcVnContainer;	(* Container with the descriptor matches (ContainerType_Vector_TcVnDMatch) *)
		ipDestImage	:	REFERENCE TO ITcVnImage;	(* Destination image (An appropriate color image will be created if required.) *)
		hrPrev	:	HRESULT;	(* HRESULT indicating the result of previous operations (If SUCCEEDED(hrPrev) equals false, no operation is executed.) *)
	END_VAR

END_FUNCTION

// Functions/Drawing/F_VN_DrawMatchesExp

	{attribute 'TcIecLibraryType'}
	{attribute 'external_name' := 'F_VN_DrawMatchesExp_GUID_B600E2B4_8A42_427F_E6C3_F8799B428051'}
	(* Draws the keypoints and matches for visualization purpose. (expert function) *)
	FUNCTION F_VN_DrawMatchesExp : HRESULT
	VAR_INPUT
		ipSrcImage1	:	ITcVnImage;	(* Source image 1 (elements of type USINT) *)
		ipKeyPoints1	:	ITcVnContainer;	(* Container with the keypoints 1 (ContainerType_Vector_TcVnKeyPoint) *)
		ipSrcImage2	:	ITcVnImage;	(* Source image 2 (elements of type USINT, must have the same number of channels as ipSrcImage1) *)
		ipKeyPoints2	:	ITcVnContainer;	(* Container with the keypoints 2 (ContainerType_Vector_TcVnKeyPoint) *)
		ipMatches1To2	:	ITcVnContainer;	(* Container with the descriptor matches (ContainerType_Vector_TcVnDMatch) *)
		ipDestImage	:	REFERENCE TO ITcVnImage;	(* Destination image (An appropriate color image will be created if required.) *)
	END_VAR
	VAR_IN_OUT
		aMatchColor	:	TcVnVector4_LREAL;	(* Color to draw the matches (for {-1, -1, -1, -1}, a random color is chosen for each point and line) *)
		aSingleColor	:	TcVnVector4_LREAL;	(* Color to draw the single keypoints (for {-1, -1, -1, -1}, a random color is chosen for each point) *)
	END_VAR
	VAR_INPUT
		ipMatchesMask	:	ITcVnContainer;	(* Mask to select the matches to be drawn (ContainerType_Vector_SINT; Set to 0 if all matches should be drawn.) *)
		eFlags	:	ETcVnDrawMatchesFlags;	(* A combination of flags to support overdrawing an existing destination image and/or drawing additional (Rich-)Keypoint information (size and orientation) and/or skipping single keypoints *)
		hrPrev	:	HRESULT;	(* HRESULT indicating the result of previous operations (If SUCCEEDED(hrPrev) equals false, no operation is executed.) *)
	END_VAR

END_FUNCTION

// Functions/Drawing/F_VN_DrawOrientation

	{attribute 'TcIecLibraryType'}
	{attribute 'external_name' := 'F_VN_DrawOrientation_GUID_FCC22671_FC88_4781_E50C_AEF3432A3647'}
	(* Draw the main axis of a set of points/contour based on a rotated rectangle. *)
	FUNCTION F_VN_DrawOrientation : HRESULT
	VAR_IN_OUT
		stOrientation	:	TcVnRotatedRectangle;	(* Rotated rectangle, containig center of mass, lenghts of axes, and rotation angle in clockwise direction *)
	END_VAR
	VAR_INPUT
		ipDestImage	:	ITcVnImage;	(* Destination image *)
	END_VAR
	VAR_IN_OUT
		aColorMainAxis	:	TcVnVector4_LREAL;	(* Color of the major axis *)
	END_VAR
	VAR_INPUT
		nThickness	:	DINT;	(* Line thickness *)
		hrPrev	:	HRESULT;	(* HRESULT indicating the result of previous operations (If SUCCEEDED(hrPrev) equals false, no operation is executed.) *)
	END_VAR

END_FUNCTION

// Functions/Drawing/F_VN_DrawOrientationExp

	{attribute 'TcIecLibraryType'}
	{attribute 'external_name' := 'F_VN_DrawOrientationExp_GUID_19F25E85_FEF4_4D6E_D101_41953AD08CA9'}
	(* Draw the main axis, the horizontal axis and the angle of a set of points/contour based on a rotated rectangle. (expert function) *)
	FUNCTION F_VN_DrawOrientationExp : HRESULT
	VAR_IN_OUT
		stOrientation	:	TcVnRotatedRectangle;	(* Rotated rectangle, containig center of mass, lenghts of axes, and rotation angle in clockwise direction *)
	END_VAR
	VAR_INPUT
		ipDestImage	:	ITcVnImage;	(* Destination image *)
	END_VAR
	VAR_IN_OUT
		aColorMainAxis	:	TcVnVector4_LREAL;	(* Color of the major axis *)
	END_VAR
	VAR_INPUT
		nThickness	:	DINT;	(* Line thickness *)
	END_VAR
	VAR_IN_OUT
		aColorHorizontalAxis	:	TcVnVector4_LREAL;	(* Color of the horizontal axis *)
	END_VAR
	VAR_INPUT
		fFontScale	:	LREAL;	(* Scaling factor for the text *)
		hrPrev	:	HRESULT;	(* HRESULT indicating the result of previous operations (If SUCCEEDED(hrPrev) equals false, no operation is executed.) *)
	END_VAR

END_FUNCTION

// Functions/Drawing/F_VN_DrawPoint

	{attribute 'TcIecLibraryType'}
	{attribute 'external_name' := 'F_VN_DrawPoint_GUID_9B879312_7DC8_44EC_C4FC_9A488EA56C09'}
	(* Draws a point. *)
	FUNCTION F_VN_DrawPoint : HRESULT
	VAR_INPUT
		nX	:	UDINT;	(* x coordinate of the point *)
		nY	:	UDINT;	(* y coordinate of the point *)
		ipDestImage	:	ITcVnImage;	(* Destination image *)
		eShape	:	ETcVnDrawShape;	(* Point shape *)
	END_VAR
	VAR_IN_OUT
		aColor	:	TcVnVector4_LREAL;	(* Color (for {-1, -1, -1, -1}, a random color is chosen) *)
	END_VAR
	VAR_INPUT
		hrPrev	:	HRESULT;	(* HRESULT indicating the result of previous operations (If SUCCEEDED(hrPrev) equals false, no operation is executed.) *)
	END_VAR

END_FUNCTION

// Functions/Drawing/F_VN_DrawPointExp

	{attribute 'TcIecLibraryType'}
	{attribute 'external_name' := 'F_VN_DrawPointExp_GUID_7C2F074E_1321_4D56_FBE3_A24CD470A1BA'}
	(* Draw a point. (expert function) *)
	FUNCTION F_VN_DrawPointExp : HRESULT
	VAR_INPUT
		nX	:	UDINT;	(* x coordinate of the point *)
		nY	:	UDINT;	(* y coordinate of the point *)
		ipDestImage	:	ITcVnImage;	(* Destination image *)
		eShape	:	ETcVnDrawShape;	(* Point shape *)
	END_VAR
	VAR_IN_OUT
		aColor	:	TcVnVector4_LREAL;	(* Color (for {-1, -1, -1, -1}, a random color is chosen) *)
	END_VAR
	VAR_INPUT
		nSize	:	UDINT;	(* Size of the shape (half width) *)
		nThickness	:	DINT;	(* Line thickness (if negative, the shape is filled if it is closed) *)
		eLineType	:	ETcVnLineType;	(* Line type *)
		hrPrev	:	HRESULT;	(* HRESULT indicating the result of previous operations (If SUCCEEDED(hrPrev) equals false, no operation is executed.) *)
	END_VAR

END_FUNCTION

// Functions/Drawing/F_VN_DrawPoints

	{attribute 'TcIecLibraryType'}
	{attribute 'external_name' := 'F_VN_DrawPoints_GUID_9656D157_1FFE_4DB4_ED49_74EB1F9D6D08'}
	(* Draw a collection of points. *)
	FUNCTION F_VN_DrawPoints : HRESULT
	VAR_INPUT
		ipPoints	:	ITcVnContainer;	(* Container with TcVnPoint2_DINT or TcVnPoint2_REAL elements *)
		ipDestImage	:	ITcVnImage;	(* Destination image *)
		eShape	:	ETcVnDrawShape;	(* Point shape *)
	END_VAR
	VAR_IN_OUT
		aColor	:	TcVnVector4_LREAL;	(* Color (for {-1, -1, -1, -1}, a random color is chosen for each point) *)
	END_VAR
	VAR_INPUT
		hrPrev	:	HRESULT;	(* HRESULT indicating the result of previous operations (If SUCCEEDED(hrPrev) equals false, no operation is executed.) *)
	END_VAR

END_FUNCTION

// Functions/Drawing/F_VN_DrawPointsExp

	{attribute 'TcIecLibraryType'}
	{attribute 'external_name' := 'F_VN_DrawPointsExp_GUID_442C7E83_1075_4FCA_FDBB_9507DF8733C1'}
	(* Draw a collection of points. (expert function) *)
	FUNCTION F_VN_DrawPointsExp : HRESULT
	VAR_INPUT
		ipPoints	:	ITcVnContainer;	(* Container with TcVnPoint2_DINT or TcVnPoint2_REAL elements *)
		ipDestImage	:	ITcVnImage;	(* Destination image *)
		eShape	:	ETcVnDrawShape;	(* Point shape *)
	END_VAR
	VAR_IN_OUT
		aColor	:	TcVnVector4_LREAL;	(* Color (for {-1, -1, -1, -1}, a random color is chosen for each point) *)
	END_VAR
	VAR_INPUT
		nSize	:	UDINT;	(* Size of the shape (half width) *)
		nThickness	:	DINT;	(* Line thickness (if negative, the shape is filled if it is closed) *)
		eLineType	:	ETcVnLineType;	(* Line type *)
		hrPrev	:	HRESULT;	(* HRESULT indicating the result of previous operations (If SUCCEEDED(hrPrev) equals false, no operation is executed.) *)
	END_VAR

END_FUNCTION

// Functions/Drawing/F_VN_DrawPolygon

	{attribute 'TcIecLibraryType'}
	{attribute 'external_name' := 'F_VN_DrawPolygon_GUID_5A5D3E88_1D24_4E33_F843_43E3010B8DAF'}
	(* Draw a pologon using collection of points. *)
	FUNCTION F_VN_DrawPolygon : HRESULT
	VAR_INPUT
		ipPoints	:	ITcVnContainer;	(* Container with TcVnPoint2_DINT, TcVnPoint2_REAL, or TcVnPoint2_LREAL elements *)
		ipDestImage	:	ITcVnImage;	(* Destination image *)
	END_VAR
	VAR_IN_OUT
		aColor	:	TcVnVector4_LREAL;	(* Color *)
	END_VAR
	VAR_INPUT
		nThickness	:	DINT;	(* Line thickness (if negative, the polygon is filled) *)
		hrPrev	:	HRESULT;	(* HRESULT indicating the result of previous operations (If SUCCEEDED(hrPrev) equals false, no operation is executed.) *)
	END_VAR

END_FUNCTION

// Functions/Drawing/F_VN_DrawPolygonExp

	{attribute 'TcIecLibraryType'}
	{attribute 'external_name' := 'F_VN_DrawPolygonExp_GUID_A7047CBF_9F9C_423A_F7B3_002BF6AD82DA'}
	(* Draw a pologon using collection of points. (expert function) *)
	FUNCTION F_VN_DrawPolygonExp : HRESULT
	VAR_INPUT
		ipPoints	:	ITcVnContainer;	(* Container with TcVnPoint2_DINT, TcVnPoint2_REAL, or TcVnPoint2_LREAL elements *)
		ipDestImage	:	ITcVnImage;	(* Destination image *)
	END_VAR
	VAR_IN_OUT
		aColor	:	TcVnVector4_LREAL;	(* Color *)
	END_VAR
	VAR_INPUT
		nThickness	:	DINT;	(* Line thickness (if negative, the shape is filled) *)
		bIsClosed	:	BOOL;	(* If it is true, the function draws a line from the last point to the first point to close the polygon. *)
		eLineType	:	ETcVnLineType;	(* Line type *)
		nShift	:	UDINT;	(* Fractional bits of the coordinates (bit shift) *)
		hrPrev	:	HRESULT;	(* HRESULT indicating the result of previous operations (If SUCCEEDED(hrPrev) equals false, no operation is executed.) *)
	END_VAR

END_FUNCTION

// Functions/Drawing/F_VN_DrawRectangle

	{attribute 'TcIecLibraryType'}
	{attribute 'external_name' := 'F_VN_DrawRectangle_GUID_BAE8C975_53F8_4DB1_E13E_FE2EB09C3A1E'}
	(* Draw a rectangle. *)
	FUNCTION F_VN_DrawRectangle : HRESULT
	VAR_INPUT
		nTopLeftX	:	UDINT;	(* x coordinate of the top left corner *)
		nTopLeftY	:	UDINT;	(* y coordinate of the top left corner *)
		nBottomRightX	:	UDINT;	(* x coordinate of the bottom right corner *)
		nBottomRightY	:	UDINT;	(* y coordinate of the bottom right corner *)
		ipDestImage	:	ITcVnImage;	(* Destination image *)
	END_VAR
	VAR_IN_OUT
		aColor	:	TcVnVector4_LREAL;	(* Color *)
	END_VAR
	VAR_INPUT
		nThickness	:	DINT;	(* Line thickness (if negative, the rectangle is filled) *)
		hrPrev	:	HRESULT;	(* HRESULT indicating the result of previous operations (If SUCCEEDED(hrPrev) equals false, no operation is executed.) *)
	END_VAR

END_FUNCTION

// Functions/Drawing/F_VN_DrawRectangle_TcVnRectangle_DINT

	{attribute 'TcIecLibraryType'}
	{attribute 'external_name' := 'F_VN_DrawRectangle_TcVnRectangle_DINT_GUID_450BE9BF_BBF1_4DA3_DBD8_FFA0FA393EC7'}
	(* Draw a rectangle. *)
	FUNCTION F_VN_DrawRectangle_TcVnRectangle_DINT : HRESULT
	VAR_IN_OUT
		stRectangle	:	TcVnRectangle_DINT;	(* Rectangle to be drawn *)
	END_VAR
	VAR_INPUT
		ipDestImage	:	ITcVnImage;	(* Destination image *)
	END_VAR
	VAR_IN_OUT
		aColor	:	TcVnVector4_LREAL;	(* Color *)
	END_VAR
	VAR_INPUT
		nThickness	:	DINT;	(* Line thickness (if negative, the rectangle is filled) *)
		hrPrev	:	HRESULT;	(* HRESULT indicating the result of previous operations (If SUCCEEDED(hrPrev) equals false, no operation is executed.) *)
	END_VAR

END_FUNCTION

// Functions/Drawing/F_VN_DrawRectangle_TcVnRectangle_UDINT

	{attribute 'TcIecLibraryType'}
	{attribute 'external_name' := 'F_VN_DrawRectangle_TcVnRectangle_UDINT_GUID_3BECEC40_2788_4F03_DFF1_146257DA9F32'}
	(* Draw a rectangle. *)
	FUNCTION F_VN_DrawRectangle_TcVnRectangle_UDINT : HRESULT
	VAR_IN_OUT
		stRectangle	:	TcVnRectangle_UDINT;	(* Rectangle to be drawn *)
	END_VAR
	VAR_INPUT
		ipDestImage	:	ITcVnImage;	(* Destination image *)
	END_VAR
	VAR_IN_OUT
		aColor	:	TcVnVector4_LREAL;	(* Color *)
	END_VAR
	VAR_INPUT
		nThickness	:	DINT;	(* Line thickness (if negative, the rectangle is filled) *)
		hrPrev	:	HRESULT;	(* HRESULT indicating the result of previous operations (If SUCCEEDED(hrPrev) equals false, no operation is executed.) *)
	END_VAR

END_FUNCTION

// Functions/Drawing/F_VN_DrawRotatedRectangle

	{attribute 'TcIecLibraryType'}
	{attribute 'external_name' := 'F_VN_DrawRotatedRectangle_GUID_99810E42_96B6_4915_EF2A_71DB4285EDBD'}
	(* Draw a rectangle. *)
	FUNCTION F_VN_DrawRotatedRectangle : HRESULT
	VAR_IN_OUT
		stRectangle	:	TcVnRotatedRectangle;	(* Rectangle to be drawn (rotation angle in degrees) *)
	END_VAR
	VAR_INPUT
		ipDestImage	:	ITcVnImage;	(* Destination image *)
	END_VAR
	VAR_IN_OUT
		aColor	:	TcVnVector4_LREAL;	(* Color *)
	END_VAR
	VAR_INPUT
		nThickness	:	DINT;	(* Line thickness (if negative, the rectangle is filled) *)
		hrPrev	:	HRESULT;	(* HRESULT indicating the result of previous operations (If SUCCEEDED(hrPrev) equals false, no operation is executed.) *)
	END_VAR

END_FUNCTION

// Functions/Drawing/F_VN_DrawRotatedRectangleExp

	{attribute 'TcIecLibraryType'}
	{attribute 'external_name' := 'F_VN_DrawRotatedRectangleExp_GUID_8E9823C7_6EA7_44E8_E495_52523A568D69'}
	(* Draw a rectangle. (expert function) *)
	FUNCTION F_VN_DrawRotatedRectangleExp : HRESULT
	VAR_IN_OUT
		stRectangle	:	TcVnRotatedRectangle;	(* Rectangle to be drawn (rotation angle in degrees) *)
	END_VAR
	VAR_INPUT
		ipDestImage	:	ITcVnImage;	(* Destination image *)
	END_VAR
	VAR_IN_OUT
		aColor	:	TcVnVector4_LREAL;	(* Color *)
	END_VAR
	VAR_INPUT
		nThickness	:	DINT;	(* Line thickness (if negative, the rectangle is filled) *)
		eLineType	:	ETcVnLineType;	(* Line type *)
		hrPrev	:	HRESULT;	(* HRESULT indicating the result of previous operations (If SUCCEEDED(hrPrev) equals false, no operation is executed.) *)
	END_VAR

END_FUNCTION

// Functions/Drawing/F_VN_FillCircle

	{attribute 'TcIecLibraryType'}
	{attribute 'external_name' := 'F_VN_FillCircle_GUID_2769CF19_1392_4D85_DC53_AFAC2A2A26DB'}
	(* Paint a filled circle. *)
	FUNCTION F_VN_FillCircle : HRESULT
	VAR_INPUT
		nCenterX	:	UDINT;	(* x coordinate of the center *)
		nCenterY	:	UDINT;	(* y coordinate of the center *)
		nRadius	:	UDINT;	(* Radius *)
		ipDestImage	:	ITcVnImage;	(* Destination image *)
	END_VAR
	VAR_IN_OUT
		aColor	:	TcVnVector4_LREAL;	(* Color *)
	END_VAR
	VAR_INPUT
		hrPrev	:	HRESULT;	(* HRESULT indicating the result of previous operations (If SUCCEEDED(hrPrev) equals false, no operation is executed.) *)
	END_VAR

END_FUNCTION

// Functions/Drawing/F_VN_FillContours

